LIN {X 0,Y 235.222,Z 369.249,A -85,B 0,C 180,E1 -19639.185,E2 -19639.185} C_VEL
LIN {X 0,Y 235.052,Z 370.546,A -85,B 0,C 180,E1 -19641.308,E2 -19641.308} C_VEL
LIN {X 0,Y 236.233,Z 373.828,A -85,B 0,C 180,E1 -19641.803,E2 -19641.803} C_VEL
LIN {X 0,Y 239.413,Z 381.749,A -85,B 0,C 180,E1 -19643.116,E2 -19643.116} C_VEL
LIN {X 0,Y 242.127,Z 390.64,A -85,B 0,C 180,E1 -19644.659,E2 -19644.659} C_VEL
LIN {X 0,Y 243.828,Z 398.514,A -85,B 0,C 180,E1 -19646.12,E2 -19646.12} C_VEL
LIN {X 0,Y 244.808,Z 405.816,A -85,B 0,C 180,E1 -19647.573,E2 -19647.573} C_VEL
LIN {X 0,Y 244.978,Z 410.229,A -85,B 0,C 180,E1 -19648.484,E2 -19648.484} C_VEL
LIN {X 0,Y 242.651,Z 419.105,A -85,B 0,C 180,E1 -19650.36,E2 -19650.36} C_VEL
LIN {X 0,Y 240.805,Z 425.868,A -85,B 0,C 180,E1 -19652.177,E2 -19652.177} C_VEL
LIN {X 0,Y 239.204,Z 431.176,A -85,B 0,C 180,E1 -19653.931,E2 -19653.931} C_VEL
LIN {X 0,Y 237.916,Z 435.038,A -85,B 0,C 180,E1 -19655.465,E2 -19655.465} C_VEL
LIN {X 0,Y 236.981,Z 437.92,A -85,B 0,C 180,E1 -19656.798,E2 -19656.798} C_VEL
LIN {X 0,Y 235.546,Z 441.794,A -85,B 0,C 180,E1 -19659.123,E2 -19659.123} C_VEL
LIN {X 0,Y 234.489,Z 444.579,A -85,B 0,C 180,E1 -19661.468,E2 -19661.468} C_VEL
LIN {X 0,Y 233.648,Z 446.359,A -85,B 0,C 180,E1 -19663.785,E2 -19663.785} C_VEL
LIN {X 0,Y 233.007,Z 447.26,A -85,B 0,C 180,E1 -19666.373,E2 -19666.373} C_VEL
LIN {X 0,Y 232.684,Z 447.05,A -85,B 0,C 180,E1 -19669.031,E2 -19669.031} C_VEL
LIN {X 0,Y 232.685,Z 445.653,A -85,B 0,C 180,E1 -19671.745,E2 -19671.745} C_VEL
LIN {X 0,Y 233.077,Z 442.082,A -85,B 0,C 180,E1 -19675.044,E2 -19675.044} C_VEL
LIN {X 0,Y 233.542,Z 438.663,A -85,B 0,C 180,E1 -19677.2,E2 -19677.2} C_VEL
LIN {X 0,Y 234.152,Z 434.313,A -85,B 0,C 180,E1 -19679.317,E2 -19679.317} C_VEL
LIN {X 0,Y 234.95,Z 428.913,A -85,B 0,C 180,E1 -19681.403,E2 -19681.403} C_VEL
LIN {X 0,Y 235.933,Z 422.286,A -85,B 0,C 180,E1 -19683.458,E2 -19683.458} C_VEL
LIN {X 0,Y 237.124,Z 413.918,A -85,B 0,C 180,E1 -19685.482,E2 -19685.482} C_VEL
LIN {X 0,Y 238.222,Z 405.62,A -85,B 0,C 180,E1 -19687.085,E2 -19687.085} C_VEL
LIN {X 0,Y 238.95,Z 398.643,A -85,B 0,C 180,E1 -19688.2,E2 -19688.2} C_VEL
LIN {X 0,Y 237.705,Z 390.04,A -85,B 0,C 180,E1 -19689.443,E2 -19689.443} C_VEL
LIN {X 0,Y 236.315,Z 381.565,A -85,B 0,C 180,E1 -19690.451,E2 -19690.451} C_VEL
LIN {X 0,Y 234.286,Z 371.556,A -85,B 0,C 180,E1 -19691.412,E2 -19691.412} C_VEL
LIN {X 0,Y 233.578,Z 368.098,A -85,B 0,C 180,E1 -19691.694,E2 -19691.694} C_VEL
LIN {X 0,Y 234.064,Z 364.147,A -85,B 0,C 180,E1 -19696.542,E2 -19696.542} C_VEL
LIN {X 0,Y 234.945,Z 364.031,A -85,B 0,C 180,E1 -19701.396,E2 -19701.396} C_VEL
LIN {X 0,Y 235.185,Z 364.002,A -85,B 0,C 180,E1 -19703.133,E2 -19703.133} C_VEL
LIN {X 0,Y 235.586,Z 363.954,A -85,B 0,C 180,E1 -19708.288,E2 -19708.288} C_VEL
LIN {X 0,Y 235.588,Z 363.952,A -85,B 0,C 180,E1 -19711.707,E2 -19711.707} C_VEL
LIN {X 0,Y 235.397,Z 363.973,A -85,B 0,C 180,E1 -19716.857,E2 -19716.857} C_VEL
LIN {X 0,Y 235.243,Z 363.992,A -85,B 0,C 180,E1 -19720.324,E2 -19720.324} C_VEL
LIN {X 0,Y 235.103,Z 364.013,A -85,B 0,C 180,E1 -19725.605,E2 -19725.605} C_VEL
LIN {X 0,Y 234.998,Z 364.023,A -85,B 0,C 180,E1 -19729.204,E2 -19729.204} C_VEL
LIN {X 0,Y 234.95,Z 364.029,A -85,B 0,C 180,E1 -19732.881,E2 -19732.881} C_VEL
LIN {X 0,Y 234.957,Z 364.027,A -85,B 0,C 180,E1 -19736.656,E2 -19736.656} C_VEL
LIN {X 0,Y 234.919,Z 364.032,A -85,B 0,C 180,E1 -19740.567,E2 -19740.567} C_VEL
LIN {X 0,Y 234.948,Z 364.029,A -85,B 0,C 180,E1 -19744.632,E2 -19744.632} C_VEL
LIN {X 0,Y 234.984,Z 364.026,A -85,B 0,C 180,E1 -19748.961,E2 -19748.961} C_VEL
LIN {X 0,Y 234.983,Z 364.024,A -85,B 0,C 180,E1 -19753.46,E2 -19753.46} C_VEL
LIN {X 0,Y 234.983,Z 364.025,A -85,B 0,C 180,E1 -19756.539,E2 -19756.539} C_VEL
LIN {X 0,Y 234.957,Z 364.029,A -85,B 0,C 180,E1 -19761.089,E2 -19761.089} C_VEL
LIN {X 0,Y 234.947,Z 364.03,A -85,B 0,C 180,E1 -19765.367,E2 -19765.367} C_VEL
LIN {X 0,Y 234.956,Z 364.028,A -85,B 0,C 180,E1 -19770.158,E2 -19770.158} C_VEL
LIN {X 0,Y 234.989,Z 364.025,A -85,B 0,C 180,E1 -19775.249,E2 -19775.249} C_VEL
LIN {X 0,Y 235.039,Z 364.016,A -85,B 0,C 180,E1 -19778.975,E2 -19778.975} C_VEL
LIN {X 0,Y 235.105,Z 364.01,A -85,B 0,C 180,E1 -19783.044,E2 -19783.044} C_VEL
LIN {X 0,Y 235.136,Z 364.006,A -85,B 0,C 180,E1 -19787.925,E2 -19787.925} C_VEL
LIN {X 0,Y 235.379,Z 363.976,A -85,B 0,C 180,E1 -19791.416,E2 -19791.416} C_VEL
LIN {X 0,Y 235.395,Z 363.973,A -85,B 0,C 180,E1 -19793.143,E2 -19793.143} C_VEL
LIN {X 0,Y 235.586,Z 363.952,A -85,B 0,C 180,E1 -19798.292,E2 -19798.292} C_VEL
LIN {X 0,Y 235.587,Z 363.952,A -85,B 0,C 180,E1 -19801.711,E2 -19801.711} C_VEL
LIN {X 0,Y 235.397,Z 363.973,A -85,B 0,C 180,E1 -19806.86,E2 -19806.86} C_VEL
LIN {X 0,Y 235.245,Z 363.992,A -85,B 0,C 180,E1 -19810.328,E2 -19810.328} C_VEL
LIN {X 0,Y 235.106,Z 364.013,A -85,B 0,C 180,E1 -19815.608,E2 -19815.608} C_VEL
LIN {X 0,Y 235.001,Z 364.024,A -85,B 0,C 180,E1 -19819.208,E2 -19819.208} C_VEL
LIN {X 0,Y 234.954,Z 364.028,A -85,B 0,C 180,E1 -19822.885,E2 -19822.885} C_VEL
LIN {X 0,Y 234.963,Z 364.028,A -85,B 0,C 180,E1 -19826.66,E2 -19826.66} C_VEL
LIN {X 0,Y 234.926,Z 364.031,A -85,B 0,C 180,E1 -19830.57,E2 -19830.57} C_VEL
LIN {X 0,Y 234.921,Z 364.034,A -85,B 0,C 180,E1 -19834.641,E2 -19834.641} C_VEL
LIN {X 0,Y 234.937,Z 364.032,A -85,B 0,C 180,E1 -19838.947,E2 -19838.947} C_VEL
LIN {X 0,Y 234.887,Z 364.037,A -85,B 0,C 180,E1 -19843.488,E2 -19843.488} C_VEL
LIN {X 0,Y 235.054,Z 364.178,A -85,B 0,C 180,E1 -19847.266,E2 -19847.266} C_VEL
LIN {X 0,Y 236.079,Z 369.576,A -85,B 0,C 180,E1 -19852.395,E2 -19852.395} C_VEL
LIN {X 0,Y 236.457,Z 371.989,A -85,B 0,C 180,E1 -19854.592,E2 -19854.592} C_VEL
LIN {X 0,Y 235.755,Z 373.624,A -85,B 0,C 180,E1 -19855.954,E2 -19855.954} C_VEL
LIN {X 0,Y 233.999,Z 375.327,A -85,B 0,C 180,E1 -19857.275,E2 -19857.275} C_VEL
LIN {X 0,Y 229.645,Z 378.781,A -85,B 0,C 180,E1 -19859.922,E2 -19859.922} C_VEL
LIN {X 0,Y 228.207,Z 380.506,A -85,B 0,C 180,E1 -19861.321,E2 -19861.321} C_VEL
LIN {X 0,Y 227.99,Z 381.073,A -85,B 0,C 180,E1 -19861.802,E2 -19861.802} C_VEL
LIN {X 0,Y 226.914,Z 387.476,A -85,B 0,C 180,E1 -19867.226,E2 -19867.226} C_VEL
LIN {X 0,Y 226.84,Z 388.158,A -85,B 0,C 180,E1 -19867.8,E2 -19867.8} C_VEL
LIN {X 0,Y 228.206,Z 400.804,A -85,B 0,C 180,E1 -19868.833,E2 -19868.833} C_VEL
LIN {X 0,Y 228.996,Z 409.707,A -85,B 0,C 180,E1 -19869.819,E2 -19869.819} C_VEL
LIN {X 0,Y 229.519,Z 418.83,A -85,B 0,C 180,E1 -19871.074,E2 -19871.074} C_VEL
LIN {X 0,Y 229.83,Z 426.888,A -85,B 0,C 180,E1 -19872.427,E2 -19872.427} C_VEL
LIN {X 0,Y 229.768,Z 431.689,A -85,B 0,C 180,E1 -19873.339,E2 -19873.339} C_VEL
LIN {X 0,Y 228.714,Z 438.58,A -85,B 0,C 180,E1 -19874.862,E2 -19874.862} C_VEL
LIN {X 0,Y 227.782,Z 445.123,A -85,B 0,C 180,E1 -19876.623,E2 -19876.623} C_VEL
LIN {X 0,Y 227.043,Z 450.571,A -85,B 0,C 180,E1 -19878.395,E2 -19878.395} C_VEL
LIN {X 0,Y 226.506,Z 455.12,A -85,B 0,C 180,E1 -19880.177,E2 -19880.177} C_VEL
LIN {X 0,Y 226.101,Z 458.892,A -85,B 0,C 180,E1 -19881.962,E2 -19881.962} C_VEL
LIN {X 0,Y 225.806,Z 463.172,A -85,B 0,C 180,E1 -19884.645,E2 -19884.645} C_VEL
LIN {X 0,Y 225.811,Z 465.347,A -85,B 0,C 180,E1 -19886.434,E2 -19886.434} C_VEL
LIN {X 0,Y 225.863,Z 466.928,A -85,B 0,C 180,E1 -19888.219,E2 -19888.219} C_VEL
LIN {X 0,Y 225.879,Z 467.899,A -85,B 0,C 180,E1 -19890.002,E2 -19890.002} C_VEL
LIN {X 0,Y 225.837,Z 468.378,A -85,B 0,C 180,E1 -19891.786,E2 -19891.786} C_VEL
LIN {X 0,Y 225.724,Z 468.081,A -85,B 0,C 180,E1 -19894.898,E2 -19894.898} C_VEL
LIN {X 0,Y 225.925,Z 466.884,A -85,B 0,C 180,E1 -19897.15,E2 -19897.15} C_VEL
LIN {X 0,Y 226.536,Z 464.45,A -85,B 0,C 180,E1 -19899.827,E2 -19899.827} C_VEL
LIN {X 0,Y 227.599,Z 460.723,A -85,B 0,C 180,E1 -19902.485,E2 -19902.485} C_VEL
LIN {X 0,Y 228.613,Z 457.567,A -85,B 0,C 180,E1 -19904.239,E2 -19904.239} C_VEL
LIN {X 0,Y 230.195,Z 452.594,A -85,B 0,C 180,E1 -19906.406,E2 -19906.406} C_VEL
LIN {X 0,Y 232.154,Z 446.383,A -85,B 0,C 180,E1 -19908.536,E2 -19908.536} C_VEL
LIN {X 0,Y 233.868,Z 440.38,A -85,B 0,C 180,E1 -19910.22,E2 -19910.22} C_VEL
LIN {X 0,Y 234.91,Z 434.608,A -85,B 0,C 180,E1 -19911.639,E2 -19911.639} C_VEL
LIN {X 0,Y 235.513,Z 426.948,A -85,B 0,C 180,E1 -19913.293,E2 -19913.293} C_VEL
LIN {X 0,Y 235.484,Z 419.713,A -85,B 0,C 180,E1 -19914.7,E2 -19914.7} C_VEL
LIN {X 0,Y 234.896,Z 411.306,A -85,B 0,C 180,E1 -19916.155,E2 -19916.155} C_VEL
LIN {X 0,Y 233.253,Z 401.765,A -85,B 0,C 180,E1 -19917.679,E2 -19917.679} C_VEL
LIN {X 0,Y 230.783,Z 391.922,A -85,B 0,C 180,E1 -19919.135,E2 -19919.135} C_VEL
LIN {X 0,Y 229.176,Z 386.225,A -85,B 0,C 180,E1 -19919.919,E2 -19919.919} C_VEL
LIN {X 0,Y 229.114,Z 385.693,A -85,B 0,C 180,E1 -19919.974,E2 -19919.974} C_VEL
LIN {X 0,Y 230.038,Z 382.099,A -85,B 0,C 180,E1 -19923.364,E2 -19923.364} C_VEL
LIN {X 0,Y 230.33,Z 380.041,A -85,B 0,C 180,E1 -19925.435,E2 -19925.435} C_VEL
LIN {X 0,Y 230.126,Z 378.022,A -85,B 0,C 180,E1 -19927.649,E2 -19927.649} C_VEL
LIN {X 0,Y 229.807,Z 375.884,A -85,B 0,C 180,E1 -19930.131,E2 -19930.131} C_VEL
LIN {X 0,Y 229.106,Z 372.001,A -85,B 0,C 180,E1 -19935.125,E2 -19935.125} C_VEL
LIN {X 0,Y 228.556,Z 368.903,A -85,B 0,C 180,E1 -19939.777,E2 -19939.777} C_VEL
LIN {X 0,Y 228.267,Z 366.929,A -85,B 0,C 180,E1 -19943.181,E2 -19943.181} C_VEL
LIN {X 0,Y 227.952,Z 365.343,A -85,B 0,C 180,E1 -19946.353,E2 -19946.353} C_VEL
LIN {X 0,Y 227.906,Z 364.908,A -85,B 0,C 180,E1 -19949.709,E2 -19949.709} C_VEL
LIN {X 0,Y 227.938,Z 364.906,A -85,B 0,C 180,E1 -19954.425,E2 -19954.425} C_VEL
LIN {X 0,Y 227.972,Z 364.9,A -85,B 0,C 180,E1 -19958.286,E2 -19958.286} C_VEL
LIN {X 0,Y 228.044,Z 364.891,A -85,B 0,C 180,E1 -19962.825,E2 -19962.825} C_VEL
LIN {X 0,Y 228.077,Z 364.887,A -85,B 0,C 180,E1 -19967.542,E2 -19967.542} C_VEL
LIN {X 0,Y 228.268,Z 364.864,A -85,B 0,C 180,E1 -19971.143,E2 -19971.143} C_VEL
LIN {X 0,Y 228.318,Z 364.859,A -85,B 0,C 180,E1 -19972.926,E2 -19972.926} C_VEL
LIN {X 0,Y 228.558,Z 364.824,A -85,B 0,C 180,E1 -19978.236,E2 -19978.236} C_VEL
LIN {X 0,Y 228.56,Z 364.825,A -85,B 0,C 180,E1 -19981.76,E2 -19981.76} C_VEL
LIN {X 0,Y 228.324,Z 364.857,A -85,B 0,C 180,E1 -19987.071,E2 -19987.071} C_VEL
LIN {X 0,Y 228.346,Z 366.209,A -85,B 0,C 180,E1 -19990.64,E2 -19990.64} C_VEL
LIN {X 0,Y 228.451,Z 367.882,A -85,B 0,C 180,E1 -19994.245,E2 -19994.245} C_VEL
LIN {X 0,Y 228.33,Z 369.822,A -85,B 0,C 180,E1 -19997.925,E2 -19997.925} C_VEL
LIN {X 0,Y 228.168,Z 371.16,A -85,B 0,C 180,E1 -19999.979,E2 -19999.979} C_VEL
LIN {X 0,Y 229.395,Z 374.35,A -85,B 0,C 180,E1 -20000.51,E2 -20000.51} C_VEL
LIN {X 0,Y 232.806,Z 382.459,A -85,B 0,C 180,E1 -20002.004,E2 -20002.004} C_VEL
LIN {X 0,Y 235.293,Z 390.144,A -85,B 0,C 180,E1 -20003.428,E2 -20003.428} C_VEL
LIN {X 0,Y 237.051,Z 397.629,A -85,B 0,C 180,E1 -20004.872,E2 -20004.872} C_VEL
LIN {X 0,Y 238.198,Z 405.563,A -85,B 0,C 180,E1 -20006.526,E2 -20006.526} C_VEL
LIN {X 0,Y 238.498,Z 411.568,A -85,B 0,C 180,E1 -20007.864,E2 -20007.864} C_VEL
LIN {X 0,Y 236.344,Z 419.358,A -85,B 0,C 180,E1 -20009.563,E2 -20009.563} C_VEL
LIN {X 0,Y 234.455,Z 425.798,A -85,B 0,C 180,E1 -20011.313,E2 -20011.313} C_VEL
LIN {X 0,Y 232.512,Z 431.916,A -85,B 0,C 180,E1 -20013.386,E2 -20013.386} C_VEL
LIN {X 0,Y 230.882,Z 436.503,A -85,B 0,C 180,E1 -20015.332,E2 -20015.332} C_VEL
LIN {X 0,Y 229.205,Z 441.046,A -85,B 0,C 180,E1 -20017.822,E2 -20017.822} C_VEL
LIN {X 0,Y 227.864,Z 444.363,A -85,B 0,C 180,E1 -20020.366,E2 -20020.366} C_VEL
LIN {X 0,Y 226.802,Z 446.504,A -85,B 0,C 180,E1 -20022.975,E2 -20022.975} C_VEL
LIN {X 0,Y 226.075,Z 447.547,A -85,B 0,C 180,E1 -20025.64,E2 -20025.64} C_VEL
LIN {X 0,Y 225.655,Z 447.49,A -85,B 0,C 180,E1 -20028.369,E2 -20028.369} C_VEL
LIN {X 0,Y 225.587,Z 446.09,A -85,B 0,C 180,E1 -20031.456,E2 -20031.456} C_VEL
LIN {X 0,Y 225.798,Z 443.719,A -85,B 0,C 180,E1 -20034.019,E2 -20034.019} C_VEL
LIN {X 0,Y 226.184,Z 441.098,A -85,B 0,C 180,E1 -20035.99,E2 -20035.99} C_VEL
LIN {X 0,Y 226.86,Z 436.252,A -85,B 0,C 180,E1 -20038.678,E2 -20038.678} C_VEL
LIN {X 0,Y 227.618,Z 431.025,A -85,B 0,C 180,E1 -20040.9,E2 -20040.9} C_VEL
LIN {X 0,Y 228.344,Z 426.452,A -85,B 0,C 180,E1 -20042.503,E2 -20042.503} C_VEL
LIN {X 0,Y 229.41,Z 419.09,A -85,B 0,C 180,E1 -20044.601,E2 -20044.601} C_VEL
LIN {X 0,Y 230.518,Z 411.603,A -85,B 0,C 180,E1 -20046.324,E2 -20046.324} C_VEL
LIN {X 0,Y 231.701,Z 402.878,A -85,B 0,C 180,E1 -20047.951,E2 -20047.951} C_VEL
LIN {X 0,Y 232.001,Z 399.711,A -85,B 0,C 180,E1 -20048.448,E2 -20048.448} C_VEL
LIN {X 0,Y 230.807,Z 391.249,A -85,B 0,C 180,E1 -20049.733,E2 -20049.733} C_VEL
LIN {X 0,Y 229.483,Z 382.947,A -85,B 0,C 180,E1 -20050.776,E2 -20050.776} C_VEL
LIN {X 0,Y 227.536,Z 373.182,A -85,B 0,C 180,E1 -20051.774,E2 -20051.774} C_VEL
LIN {X 0,Y 226.56,Z 368.36,A -85,B 0,C 180,E1 -20052.218,E2 -20052.218} C_VEL
LIN {X 0,Y 227.018,Z 365.024,A -85,B 0,C 180,E1 -20056.572,E2 -20056.572} C_VEL
LIN {X 0,Y 227.87,Z 364.912,A -85,B 0,C 180,E1 -20061.127,E2 -20061.127} C_VEL
LIN {X 0,Y 228.099,Z 364.885,A -85,B 0,C 180,E1 -20062.918,E2 -20062.918} C_VEL
LIN {X 0,Y 228.544,Z 364.832,A -85,B 0,C 180,E1 -20068.236,E2 -20068.236} C_VEL
LIN {X 0,Y 228.547,Z 364.83,A -85,B 0,C 180,E1 -20071.76,E2 -20071.76} C_VEL
LIN {X 0,Y 228.349,Z 364.851,A -85,B 0,C 180,E1 -20077.069,E2 -20077.069} C_VEL
LIN {X 0,Y 228.162,Z 364.873,A -85,B 0,C 180,E1 -20080.648,E2 -20080.648} C_VEL
LIN {X 0,Y 228.047,Z 364.891,A -85,B 0,C 180,E1 -20086.1,E2 -20086.1} C_VEL
LIN {X 0,Y 227.932,Z 364.904,A -85,B 0,C 180,E1 -20089.824,E2 -20089.824} C_VEL
LIN {X 0,Y 227.903,Z 364.911,A -85,B 0,C 180,E1 -20093.631,E2 -20093.631} C_VEL
LIN {X 0,Y 227.873,Z 364.911,A -85,B 0,C 180,E1 -20097.554,E2 -20097.554} C_VEL
LIN {X 0,Y 227.86,Z 364.915,A -85,B 0,C 180,E1 -20101.621,E2 -20101.621} C_VEL
LIN {X 0,Y 227.89,Z 364.906,A -85,B 0,C 180,E1 -20105.867,E2 -20105.867} C_VEL
LIN {X 0,Y 227.905,Z 364.907,A -85,B 0,C 180,E1 -20110.356,E2 -20110.356} C_VEL
LIN {X 0,Y 227.907,Z 364.907,A -85,B 0,C 180,E1 -20114.829,E2 -20114.829} C_VEL
LIN {X 0,Y 227.922,Z 364.905,A -85,B 0,C 180,E1 -20117.731,E2 -20117.731} C_VEL
LIN {X 0,Y 227.868,Z 364.91,A -85,B 0,C 180,E1 -20121.916,E2 -20121.916} C_VEL
LIN {X 0,Y 227.877,Z 364.911,A -85,B 0,C 180,E1 -20126.373,E2 -20126.373} C_VEL
LIN {X 0,Y 227.906,Z 364.908,A -85,B 0,C 180,E1 -20130.438,E2 -20130.438} C_VEL
LIN {X 0,Y 227.922,Z 364.907,A -85,B 0,C 180,E1 -20134.427,E2 -20134.427} C_VEL
LIN {X 0,Y 227.999,Z 364.897,A -85,B 0,C 180,E1 -20138.293,E2 -20138.293} C_VEL
LIN {X 0,Y 228.034,Z 364.892,A -85,B 0,C 180,E1 -20142.818,E2 -20142.818} C_VEL
LIN {X 0,Y 228.083,Z 364.882,A -85,B 0,C 180,E1 -20147.546,E2 -20147.546} C_VEL
LIN {X 0,Y 228.314,Z 364.856,A -85,B 0,C 180,E1 -20151.148,E2 -20151.148} C_VEL
LIN {X 0,Y 228.347,Z 364.852,A -85,B 0,C 180,E1 -20152.93,E2 -20152.93} C_VEL
LIN {X 0,Y 228.545,Z 364.829,A -85,B 0,C 180,E1 -20158.24,E2 -20158.24} C_VEL
LIN {X 0,Y 228.546,Z 364.83,A -85,B 0,C 180,E1 -20161.764,E2 -20161.764} C_VEL
LIN {X 0,Y 228.349,Z 364.851,A -85,B 0,C 180,E1 -20167.073,E2 -20167.073} C_VEL
LIN {X 0,Y 228.159,Z 364.874,A -85,B 0,C 180,E1 -20170.652,E2 -20170.652} C_VEL
LIN {X 0,Y 228.057,Z 364.887,A -85,B 0,C 180,E1 -20174.274,E2 -20174.274} C_VEL
LIN {X 0,Y 227.996,Z 364.896,A -85,B 0,C 180,E1 -20177.956,E2 -20177.956} C_VEL
LIN {X 0,Y 227.923,Z 364.903,A -85,B 0,C 180,E1 -20182.332,E2 -20182.332} C_VEL
LIN {X 0,Y 227.937,Z 364.903,A -85,B 0,C 180,E1 -20186.605,E2 -20186.605} C_VEL
LIN {X 0,Y 227.903,Z 364.905,A -85,B 0,C 180,E1 -20190.299,E2 -20190.299} C_VEL
LIN {X 0,Y 227.871,Z 364.912,A -85,B 0,C 180,E1 -20193.723,E2 -20193.723} C_VEL
LIN {X 0,Y 227.839,Z 364.913,A -85,B 0,C 180,E1 -20198.094,E2 -20198.094} C_VEL
LIN {X 0,Y 227.809,Z 364.921,A -85,B 0,C 180,E1 -20202.745,E2 -20202.745} C_VEL
LIN {X 0,Y 228.01,Z 365.07,A -85,B 0,C 180,E1 -20207.116,E2 -20207.116} C_VEL
LIN {X 0,Y 228.965,Z 370.174,A -85,B 0,C 180,E1 -20212.132,E2 -20212.132} C_VEL
LIN {X 0,Y 229.383,Z 372.742,A -85,B 0,C 180,E1 -20214.543,E2 -20214.543} C_VEL
LIN {X 0,Y 229.319,Z 374.955,A -85,B 0,C 180,E1 -20216.523,E2 -20216.523} C_VEL
LIN {X 0,Y 228.666,Z 378.252,A -85,B 0,C 180,E1 -20219.383,E2 -20219.383} C_VEL
LIN {X 0,Y 227.99,Z 381.073,A -85,B 0,C 180,E1 -20221.802,E2 -20221.802} C_VEL
LIN {X 0,Y 227.071,Z 382.206,A -85,B 0,C 180,E1 -20222.731,E2 -20222.731} C_VEL
LIN {X 0,Y 223.903,Z 384.061,A -85,B 0,C 180,E1 -20224.164,E2 -20224.164} C_VEL
LIN {X 0,Y 220.762,Z 385.925,A -85,B 0,C 180,E1 -20225.635,E2 -20225.635} C_VEL
LIN {X 0,Y 219.924,Z 387.076,A -85,B 0,C 180,E1 -20226.607,E2 -20226.607} C_VEL
LIN {X 0,Y 219.813,Z 387.82,A -85,B 0,C 180,E1 -20227.255,E2 -20227.255} C_VEL
LIN {X 0,Y 221.23,Z 400.594,A -85,B 0,C 180,E1 -20228.37,E2 -20228.37} C_VEL
LIN {X 0,Y 221.994,Z 409.762,A -85,B 0,C 180,E1 -20229.428,E2 -20229.428} C_VEL
LIN {X 0,Y 222.418,Z 418.033,A -85,B 0,C 180,E1 -20230.597,E2 -20230.597} C_VEL
LIN {X 0,Y 222.746,Z 425.393,A -85,B 0,C 180,E1 -20231.849,E2 -20231.849} C_VEL
LIN {X 0,Y 222.753,Z 431.444,A -85,B 0,C 180,E1 -20233.034,E2 -20233.034} C_VEL
LIN {X 0,Y 221.554,Z 439.172,A -85,B 0,C 180,E1 -20234.831,E2 -20234.831} C_VEL
LIN {X 0,Y 220.638,Z 445.564,A -85,B 0,C 180,E1 -20236.65,E2 -20236.65} C_VEL
LIN {X 0,Y 219.879,Z 450.875,A -85,B 0,C 180,E1 -20238.479,E2 -20238.479} C_VEL
LIN {X 0,Y 219.275,Z 456.267,A -85,B 0,C 180,E1 -20240.781,E2 -20240.781} C_VEL
LIN {X 0,Y 218.935,Z 459.744,A -85,B 0,C 180,E1 -20242.625,E2 -20242.625} C_VEL
LIN {X 0,Y 218.709,Z 463.215,A -85,B 0,C 180,E1 -20244.987,E2 -20244.987} C_VEL
LIN {X 0,Y 218.714,Z 464.816,A -85,B 0,C 180,E1 -20246.318,E2 -20246.318} C_VEL
LIN {X 0,Y 218.795,Z 466.416,A -85,B 0,C 180,E1 -20248.162,E2 -20248.162} C_VEL
LIN {X 0,Y 218.81,Z 467.454,A -85,B 0,C 180,E1 -20250.002,E2 -20250.002} C_VEL
LIN {X 0,Y 218.743,Z 468.003,A -85,B 0,C 180,E1 -20251.844,E2 -20251.844} C_VEL
LIN {X 0,Y 218.623,Z 467.847,A -85,B 0,C 180,E1 -20254.748,E2 -20254.748} C_VEL
LIN {X 0,Y 218.862,Z 466.661,A -85,B 0,C 180,E1 -20257.382,E2 -20257.382} C_VEL
LIN {X 0,Y 219.248,Z 465.19,A -85,B 0,C 180,E1 -20259.225,E2 -20259.225} C_VEL
LIN {X 0,Y 220.222,Z 462.044,A -85,B 0,C 180,E1 -20261.974,E2 -20261.974} C_VEL
LIN {X 0,Y 221.724,Z 457.649,A -85,B 0,C 180,E1 -20264.692,E2 -20264.692} C_VEL
LIN {X 0,Y 223.729,Z 451.653,A -85,B 0,C 180,E1 -20267.365,E2 -20267.365} C_VEL
LIN {X 0,Y 225.915,Z 445.318,A -85,B 0,C 180,E1 -20269.54,E2 -20269.54} C_VEL
LIN {X 0,Y 227.601,Z 439.223,A -85,B 0,C 180,E1 -20271.276,E2 -20271.276} C_VEL
LIN {X 0,Y 228.523,Z 433.646,A -85,B 0,C 180,E1 -20272.685,E2 -20272.685} C_VEL
LIN {X 0,Y 229.124,Z 425.632,A -85,B 0,C 180,E1 -20274.464,E2 -20274.464} C_VEL
LIN {X 0,Y 228.971,Z 417.582,A -85,B 0,C 180,E1 -20276.059,E2 -20276.059} C_VEL
LIN {X 0,Y 228.147,Z 409.462,A -85,B 0,C 180,E1 -20277.523,E2 -20277.523} C_VEL
LIN {X 0,Y 226.749,Z 401.44,A -85,B 0,C 180,E1 -20278.882,E2 -20278.882} C_VEL
LIN {X 0,Y 224.445,Z 392.356,A -85,B 0,C 180,E1 -20280.335,E2 -20280.335} C_VEL
LIN {X 0,Y 223.067,Z 387.959,A -85,B 0,C 180,E1 -20281.04,E2 -20281.04} C_VEL
LIN {X 0,Y 222.454,Z 385.249,A -85,B 0,C 180,E1 -20281.397,E2 -20281.397} C_VEL
LIN {X 0,Y 223.247,Z 382.117,A -85,B 0,C 180,E1 -20284.52,E2 -20284.52} C_VEL
LIN {X 0,Y 223.078,Z 378.973,A -85,B 0,C 180,E1 -20288.035,E2 -20288.035} C_VEL
LIN {X 0,Y 222.606,Z 376.133,A -85,B 0,C 180,E1 -20291.532,E2 -20291.532} C_VEL
LIN {X 0,Y 222.029,Z 372.99,A -85,B 0,C 180,E1 -20295.861,E2 -20295.861} C_VEL
LIN {X 0,Y 221.571,Z 369.972,A -85,B 0,C 180,E1 -20300.624,E2 -20300.624} C_VEL
LIN {X 0,Y 221.397,Z 368.697,A -85,B 0,C 180,E1 -20302.904,E2 -20302.904} C_VEL
LIN {X 0,Y 220.961,Z 366.628,A -85,B 0,C 180,E1 -20307.266,E2 -20307.266} C_VEL
LIN {X 0,Y 220.844,Z 365.789,A -85,B 0,C 180,E1 -20309.389,E2 -20309.389} C_VEL
LIN {X 0,Y 220.904,Z 365.781,A -85,B 0,C 180,E1 -20313.549,E2 -20313.549} C_VEL
LIN {X 0,Y 220.888,Z 365.784,A -85,B 0,C 180,E1 -20317.553,E2 -20317.553} C_VEL
LIN {X 0,Y 220.994,Z 365.769,A -85,B 0,C 180,E1 -20322.57,E2 -20322.57} C_VEL
LIN {X 0,Y 221.017,Z 365.767,A -85,B 0,C 180,E1 -20327.137,E2 -20327.137} C_VEL
LIN {X 0,Y 221.207,Z 365.743,A -85,B 0,C 180,E1 -20330.858,E2 -20330.858} C_VEL
LIN {X 0,Y 221.133,Z 365.754,A -85,B 0,C 180,E1 -20334.527,E2 -20334.527} C_VEL
LIN {X 0,Y 221.516,Z 365.701,A -85,B 0,C 180,E1 -20338.18,E2 -20338.18} C_VEL
LIN {X 0,Y 221.518,Z 365.703,A -85,B 0,C 180,E1 -20341.816,E2 -20341.816} C_VEL
LIN {X 0,Y 221.141,Z 365.75,A -85,B 0,C 180,E1 -20345.469,E2 -20345.469} C_VEL
LIN {X 0,Y 221.349,Z 366.292,A -85,B 0,C 180,E1 -20347.295,E2 -20347.295} C_VEL
LIN {X 0,Y 221.402,Z 367.783,A -85,B 0,C 180,E1 -20350.978,E2 -20350.978} C_VEL
LIN {X 0,Y 221.476,Z 369.468,A -85,B 0,C 180,E1 -20354.704,E2 -20354.704} C_VEL
LIN {X 0,Y 221.277,Z 371.427,A -85,B 0,C 180,E1 -20358.468,E2 -20358.468} C_VEL
LIN {X 0,Y 222.475,Z 374.707,A -85,B 0,C 180,E1 -20359.071,E2 -20359.071} C_VEL
LIN {X 0,Y 225.705,Z 381.835,A -85,B 0,C 180,E1 -20360.504,E2 -20360.504} C_VEL
LIN {X 0,Y 228.504,Z 389.954,A -85,B 0,C 180,E1 -20362.131,E2 -20362.131} C_VEL
LIN {X 0,Y 230.555,Z 398.263,A -85,B 0,C 180,E1 -20363.862,E2 -20363.862} C_VEL
LIN {X 0,Y 231.717,Z 406.222,A -85,B 0,C 180,E1 -20365.605,E2 -20365.605} C_VEL
LIN {X 0,Y 232.032,Z 413.115,A -85,B 0,C 180,E1 -20367.24,E2 -20367.24} C_VEL
LIN {X 0,Y 230.006,Z 419.935,A -85,B 0,C 180,E1 -20368.782,E2 -20368.782} C_VEL
LIN {X 0,Y 228.178,Z 425.792,A -85,B 0,C 180,E1 -20370.408,E2 -20370.408} C_VEL
LIN {X 0,Y 226.305,Z 431.357,A -85,B 0,C 180,E1 -20372.302,E2 -20372.302} C_VEL
LIN {X 0,Y 224.548,Z 436.08,A -85,B 0,C 180,E1 -20374.287,E2 -20374.287} C_VEL
LIN {X 0,Y 223.19,Z 439.612,A -85,B 0,C 180,E1 -20376.123,E2 -20376.123} C_VEL
LIN {X 0,Y 221.585,Z 443.313,A -85,B 0,C 180,E1 -20378.653,E2 -20378.653} C_VEL
LIN {X 0,Y 220.822,Z 445.045,A -85,B 0,C 180,E1 -20380.193,E2 -20380.193} C_VEL
LIN {X 0,Y 219.807,Z 446.922,A -85,B 0,C 180,E1 -20382.657,E2 -20382.657} C_VEL
LIN {X 0,Y 219.1,Z 447.876,A -85,B 0,C 180,E1 -20385.112,E2 -20385.112} C_VEL
LIN {X 0,Y 218.632,Z 447.926,A -85,B 0,C 180,E1 -20387.672,E2 -20387.672} C_VEL
LIN {X 0,Y 218.449,Z 446.85,A -85,B 0,C 180,E1 -20390.542,E2 -20390.542} C_VEL
LIN {X 0,Y 218.626,Z 444.524,A -85,B 0,C 180,E1 -20393.477,E2 -20393.477} C_VEL
LIN {X 0,Y 219.166,Z 440.644,A -85,B 0,C 180,E1 -20396.481,E2 -20396.481} C_VEL
LIN {X 0,Y 219.743,Z 436.737,A -85,B 0,C 180,E1 -20398.684,E2 -20398.684} C_VEL
LIN {X 0,Y 220.529,Z 431.478,A -85,B 0,C 180,E1 -20401,E2 -20401} C_VEL
LIN {X 0,Y 221.338,Z 426.62,A -85,B 0,C 180,E1 -20402.751,E2 -20402.751} C_VEL
LIN {X 0,Y 222.304,Z 419.915,A -85,B 0,C 180,E1 -20404.733,E2 -20404.733} C_VEL
LIN {X 0,Y 223.422,Z 412.866,A -85,B 0,C 180,E1 -20406.433,E2 -20406.433} C_VEL
LIN {X 0,Y 224.45,Z 405.347,A -85,B 0,C 180,E1 -20407.927,E2 -20407.927} C_VEL
LIN {X 0,Y 225.017,Z 400.819,A -85,B 0,C 180,E1 -20408.708,E2 -20408.708} C_VEL
LIN {X 0,Y 223.911,Z 392.463,A -85,B 0,C 180,E1 -20410.039,E2 -20410.039} C_VEL
LIN {X 0,Y 222.654,Z 384.338,A -85,B 0,C 180,E1 -20411.121,E2 -20411.121} C_VEL
LIN {X 0,Y 220.778,Z 374.728,A -85,B 0,C 180,E1 -20412.156,E2 -20412.156} C_VEL
LIN {X 0,Y 219.529,Z 368.694,A -85,B 0,C 180,E1 -20412.712,E2 -20412.712} C_VEL
LIN {X 0,Y 219.934,Z 365.908,A -85,B 0,C 180,E1 -20416.367,E2 -20416.367} C_VEL
LIN {X 0,Y 220.763,Z 365.799,A -85,B 0,C 180,E1 -20420.839,E2 -20420.839} C_VEL
LIN {X 0,Y 221.018,Z 365.768,A -85,B 0,C 180,E1 -20422.69,E2 -20422.69} C_VEL
LIN {X 0,Y 221.501,Z 365.71,A -85,B 0,C 180,E1 -20428.179,E2 -20428.179} C_VEL
LIN {X 0,Y 221.505,Z 365.707,A -85,B 0,C 180,E1 -20431.816,E2 -20431.816} C_VEL
LIN {X 0,Y 221.302,Z 365.73,A -85,B 0,C 180,E1 -20437.296,E2 -20437.296} C_VEL
LIN {X 0,Y 221.107,Z 365.751,A -85,B 0,C 180,E1 -20440.992,E2 -20440.992} C_VEL
LIN {X 0,Y 221.006,Z 365.766,A -85,B 0,C 180,E1 -20446.628,E2 -20446.628} C_VEL
LIN {X 0,Y 220.882,Z 365.779,A -85,B 0,C 180,E1 -20450.484,E2 -20450.484} C_VEL
LIN {X 0,Y 220.856,Z 365.785,A -85,B 0,C 180,E1 -20454.433,E2 -20454.433} C_VEL
LIN {X 0,Y 220.824,Z 365.786,A -85,B 0,C 180,E1 -20458.512,E2 -20458.512} C_VEL
LIN {X 0,Y 220.812,Z 365.791,A -85,B 0,C 180,E1 -20462.754,E2 -20462.754} C_VEL
LIN {X 0,Y 220.855,Z 365.786,A -85,B 0,C 180,E1 -20467.297,E2 -20467.297} C_VEL
LIN {X 0,Y 220.866,Z 365.783,A -85,B 0,C 180,E1 -20471.927,E2 -20471.927} C_VEL
LIN {X 0,Y 220.862,Z 365.783,A -85,B 0,C 180,E1 -20475.572,E2 -20475.572} C_VEL
LIN {X 0,Y 220.848,Z 365.786,A -85,B 0,C 180,E1 -20479.791,E2 -20479.791} C_VEL
LIN {X 0,Y 220.826,Z 365.789,A -85,B 0,C 180,E1 -20482.796,E2 -20482.796} C_VEL
LIN {X 0,Y 220.811,Z 365.791,A -85,B 0,C 180,E1 -20487.246,E2 -20487.246} C_VEL
LIN {X 0,Y 220.824,Z 365.786,A -85,B 0,C 180,E1 -20491.487,E2 -20491.487} C_VEL
LIN {X 0,Y 220.871,Z 365.783,A -85,B 0,C 180,E1 -20495.568,E2 -20495.568} C_VEL
LIN {X 0,Y 220.914,Z 365.774,A -85,B 0,C 180,E1 -20499.518,E2 -20499.518} C_VEL
LIN {X 0,Y 221.014,Z 365.765,A -85,B 0,C 180,E1 -20503.372,E2 -20503.372} C_VEL
LIN {X 0,Y 221.106,Z 365.752,A -85,B 0,C 180,E1 -20509.008,E2 -20509.008} C_VEL
LIN {X 0,Y 221.3,Z 365.73,A -85,B 0,C 180,E1 -20512.704,E2 -20512.704} C_VEL
LIN {X 0,Y 221.503,Z 365.707,A -85,B 0,C 180,E1 -20518.184,E2 -20518.184} C_VEL
LIN {X 0,Y 221.504,Z 365.707,A -85,B 0,C 180,E1 -20521.82,E2 -20521.82} C_VEL
LIN {X 0,Y 221.302,Z 365.73,A -85,B 0,C 180,E1 -20527.3,E2 -20527.3} C_VEL
LIN {X 0,Y 221.103,Z 365.753,A -85,B 0,C 180,E1 -20530.996,E2 -20530.996} C_VEL
LIN {X 0,Y 221.009,Z 365.766,A -85,B 0,C 180,E1 -20536.632,E2 -20536.632} C_VEL
LIN {X 0,Y 220.885,Z 365.778,A -85,B 0,C 180,E1 -20540.488,E2 -20540.488} C_VEL
LIN {X 0,Y 220.861,Z 365.784,A -85,B 0,C 180,E1 -20544.437,E2 -20544.437} C_VEL
LIN {X 0,Y 220.831,Z 365.786,A -85,B 0,C 180,E1 -20548.516,E2 -20548.516} C_VEL
LIN {X 0,Y 220.812,Z 365.792,A -85,B 0,C 180,E1 -20552.759,E2 -20552.759} C_VEL
LIN {X 0,Y 220.805,Z 365.791,A -85,B 0,C 180,E1 -20557.281,E2 -20557.281} C_VEL
LIN {X 0,Y 220.767,Z 365.796,A -85,B 0,C 180,E1 -20561.955,E2 -20561.955} C_VEL
LIN {X 0,Y 220.945,Z 365.985,A -85,B 0,C 180,E1 -20567.023,E2 -20567.023} C_VEL
LIN {X 0,Y 221.588,Z 369.531,A -85,B 0,C 180,E1 -20570.633,E2 -20570.633} C_VEL
LIN {X 0,Y 222.309,Z 373.175,A -85,B 0,C 180,E1 -20574.212,E2 -20574.212} C_VEL
LIN {X 0,Y 222.267,Z 375.535,A -85,B 0,C 180,E1 -20576.407,E2 -20576.407} C_VEL
LIN {X 0,Y 221.23,Z 380.117,A -85,B 0,C 180,E1 -20580.504,E2 -20580.504} C_VEL
LIN {X 0,Y 220.088,Z 385.78,A -85,B 0,C 180,E1 -20585.476,E2 -20585.476} C_VEL
LIN {X 0,Y 219.924,Z 387.076,A -85,B 0,C 180,E1 -20586.607,E2 -20586.607} C_VEL
LIN {X 0,Y 219.839,Z 388.555,A -85,B 0,C 180,E1 -20587.121,E2 -20587.121} C_VEL
LIN {X 0,Y 219.734,Z 391.899,A -85,B 0,C 180,E1 -20587.534,E2 -20587.534} C_VEL
LIN {X 0,Y 218.798,Z 401.426,A -85,B 0,C 180,E1 -20588.28,E2 -20588.28} C_VEL
LIN {X 0,Y 215.763,Z 412.226,A -85,B 0,C 180,E1 -20589.32,E2 -20589.32} C_VEL
LIN {X 0,Y 215.338,Z 415.796,A -85,B 0,C 180,E1 -20589.865,E2 -20589.865} C_VEL
LIN {X 0,Y 215.705,Z 425.143,A -85,B 0,C 180,E1 -20591.481,E2 -20591.481} C_VEL
LIN {X 0,Y 215.624,Z 432.219,A -85,B 0,C 180,E1 -20592.944,E2 -20592.944} C_VEL
LIN {X 0,Y 214.397,Z 439.76,A -85,B 0,C 180,E1 -20594.8,E2 -20594.8} C_VEL
LIN {X 0,Y 213.504,Z 445.999,A -85,B 0,C 180,E1 -20596.681,E2 -20596.681} C_VEL
LIN {X 0,Y 212.742,Z 451.171,A -85,B 0,C 180,E1 -20598.57,E2 -20598.57} C_VEL
LIN {X 0,Y 212.247,Z 455.484,A -85,B 0,C 180,E1 -20600.473,E2 -20600.473} C_VEL
LIN {X 0,Y 211.786,Z 460.566,A -85,B 0,C 180,E1 -20603.333,E2 -20603.333} C_VEL
LIN {X 0,Y 211.621,Z 464.24,A -85,B 0,C 180,E1 -20606.194,E2 -20606.194} C_VEL
LIN {X 0,Y 211.726,Z 465.884,A -85,B 0,C 180,E1 -20608.1,E2 -20608.1} C_VEL
LIN {X 0,Y 211.743,Z 466.999,A -85,B 0,C 180,E1 -20610.002,E2 -20610.002} C_VEL
LIN {X 0,Y 211.65,Z 467.624,A -85,B 0,C 180,E1 -20611.905,E2 -20611.905} C_VEL
LIN {X 0,Y 211.54,Z 467.604,A -85,B 0,C 180,E1 -20614.648,E2 -20614.648} C_VEL
LIN {X 0,Y 211.823,Z 466.441,A -85,B 0,C 180,E1 -20617.629,E2 -20617.629} C_VEL
LIN {X 0,Y 212.234,Z 465.051,A -85,B 0,C 180,E1 -20619.533,E2 -20619.533} C_VEL
LIN {X 0,Y 213.276,Z 461.989,A -85,B 0,C 180,E1 -20622.37,E2 -20622.37} C_VEL
LIN {X 0,Y 214.847,Z 457.704,A -85,B 0,C 180,E1 -20625.173,E2 -20625.173} C_VEL
LIN {X 0,Y 216.974,Z 451.937,A -85,B 0,C 180,E1 -20627.924,E2 -20627.924} C_VEL
LIN {X 0,Y 219.266,Z 445.758,A -85,B 0,C 180,E1 -20630.157,E2 -20630.157} C_VEL
LIN {X 0,Y 221.022,Z 439.816,A -85,B 0,C 180,E1 -20631.942,E2 -20631.942} C_VEL
LIN {X 0,Y 222.18,Z 432.74,A -85,B 0,C 180,E1 -20633.795,E2 -20633.795} C_VEL
LIN {X 0,Y 222.671,Z 425.486,A -85,B 0,C 180,E1 -20635.472,E2 -20635.472} C_VEL
LIN {X 0,Y 222.576,Z 417.744,A -85,B 0,C 180,E1 -20637.09,E2 -20637.09} C_VEL
LIN {X 0,Y 221.813,Z 409.714,A -85,B 0,C 180,E1 -20638.638,E2 -20638.638} C_VEL
LIN {X 0,Y 220.396,Z 401.474,A -85,B 0,C 180,E1 -20640.119,E2 -20640.119} C_VEL
LIN {X 0,Y 217.787,Z 391.561,A -85,B 0,C 180,E1 -20641.836,E2 -20641.836} C_VEL
LIN {X 0,Y 216.715,Z 388.139,A -85,B 0,C 180,E1 -20642.438,E2 -20642.438} C_VEL
LIN {X 0,Y 215.865,Z 384.791,A -85,B 0,C 180,E1 -20642.953,E2 -20642.953} C_VEL
LIN {X 0,Y 216.262,Z 382.162,A -85,B 0,C 180,E1 -20645.803,E2 -20645.803} C_VEL
LIN {X 0,Y 216.02,Z 379.764,A -85,B 0,C 180,E1 -20648.663,E2 -20648.663} C_VEL
LIN {X 0,Y 215.411,Z 376.28,A -85,B 0,C 180,E1 -20653.25,E2 -20653.25} C_VEL
LIN {X 0,Y 215.007,Z 373.97,A -85,B 0,C 180,E1 -20656.65,E2 -20656.65} C_VEL
LIN {X 0,Y 214.531,Z 370.884,A -85,B 0,C 180,E1 -20661.838,E2 -20661.838} C_VEL
LIN {X 0,Y 214.163,Z 368.805,A -85,B 0,C 180,E1 -20666.089,E2 -20666.089} C_VEL
LIN {X 0,Y 213.825,Z 367.081,A -85,B 0,C 180,E1 -20670.459,E2 -20670.459} C_VEL
LIN {X 0,Y 213.836,Z 366.661,A -85,B 0,C 180,E1 -20672.603,E2 -20672.603} C_VEL
LIN {X 0,Y 213.862,Z 366.658,A -85,B 0,C 180,E1 -20676.952,E2 -20676.952} C_VEL
LIN {X 0,Y 213.953,Z 366.646,A -85,B 0,C 180,E1 -20682.803,E2 -20682.803} C_VEL
LIN {X 0,Y 213.96,Z 366.647,A -85,B 0,C 180,E1 -20686.705,E2 -20686.705} C_VEL
LIN {X 0,Y 214.145,Z 366.623,A -85,B 0,C 180,E1 -20690.554,E2 -20690.554} C_VEL
LIN {X 0,Y 214.095,Z 366.631,A -85,B 0,C 180,E1 -20694.347,E2 -20694.347} C_VEL
LIN {X 0,Y 214.449,Z 366.581,A -85,B 0,C 180,E1 -20698.12,E2 -20698.12} C_VEL
LIN {X 0,Y 214.554,Z 366.573,A -85,B 0,C 180,E1 -20699.998,E2 -20699.998} C_VEL
LIN {X 0,Y 214.451,Z 366.583,A -85,B 0,C 180,E1 -20701.876,E2 -20701.876} C_VEL
LIN {X 0,Y 214.148,Z 366.671,A -85,B 0,C 180,E1 -20703.762,E2 -20703.762} C_VEL
LIN {X 0,Y 214.402,Z 367.886,A -85,B 0,C 180,E1 -20707.532,E2 -20707.532} C_VEL
LIN {X 0,Y 214.45,Z 369.358,A -85,B 0,C 180,E1 -20711.338,E2 -20711.338} C_VEL
LIN {X 0,Y 214.48,Z 371.085,A -85,B 0,C 180,E1 -20715.195,E2 -20715.195} C_VEL
LIN {X 0,Y 214.436,Z 371.869,A -85,B 0,C 180,E1 -20716.847,E2 -20716.847} C_VEL
LIN {X 0,Y 215.468,Z 374.789,A -85,B 0,C 180,E1 -20717.4,E2 -20717.4} C_VEL
LIN {X 0,Y 216.696,Z 377.143,A -85,B 0,C 180,E1 -20717.956,E2 -20717.956} C_VEL
LIN {X 0,Y 220.293,Z 385.578,A -85,B 0,C 180,E1 -20719.83,E2 -20719.83} C_VEL
LIN {X 0,Y 222.773,Z 393.314,A -85,B 0,C 180,E1 -20721.513,E2 -20721.513} C_VEL
LIN {X 0,Y 224.668,Z 402.194,A -85,B 0,C 180,E1 -20723.504,E2 -20723.504} C_VEL
LIN {X 0,Y 225.612,Z 410.864,A -85,B 0,C 180,E1 -20725.59,E2 -20725.59} C_VEL
LIN {X 0,Y 225.55,Z 414.792,A -85,B 0,C 180,E1 -20726.608,E2 -20726.608} C_VEL
LIN {X 0,Y 223.389,Z 421.606,A -85,B 0,C 180,E1 -20728.245,E2 -20728.245} C_VEL
LIN {X 0,Y 221.316,Z 427.751,A -85,B 0,C 180,E1 -20730.077,E2 -20730.077} C_VEL
LIN {X 0,Y 218.876,Z 434.365,A -85,B 0,C 180,E1 -20732.552,E2 -20732.552} C_VEL
LIN {X 0,Y 216.794,Z 439.382,A -85,B 0,C 180,E1 -20735.057,E2 -20735.057} C_VEL
LIN {X 0,Y 215.449,Z 442.421,A -85,B 0,C 180,E1 -20737.004,E2 -20737.004} C_VEL
LIN {X 0,Y 213.978,Z 445.395,A -85,B 0,C 180,E1 -20739.629,E2 -20739.629} C_VEL
LIN {X 0,Y 213.233,Z 446.7,A -85,B 0,C 180,E1 -20741.235,E2 -20741.235} C_VEL
LIN {X 0,Y 212.279,Z 448.115,A -85,B 0,C 180,E1 -20744.044,E2 -20744.044} C_VEL
LIN {X 0,Y 211.647,Z 448.363,A -85,B 0,C 180,E1 -20746.928,E2 -20746.928} C_VEL
LIN {X 0,Y 211.376,Z 447.436,A -85,B 0,C 180,E1 -20749.878,E2 -20749.878} C_VEL
LIN {X 0,Y 211.528,Z 444.942,A -85,B 0,C 180,E1 -20753.267,E2 -20753.267} C_VEL
LIN {X 0,Y 211.97,Z 441.717,A -85,B 0,C 180,E1 -20755.98,E2 -20755.98} C_VEL
LIN {X 0,Y 212.631,Z 437.195,A -85,B 0,C 180,E1 -20758.676,E2 -20758.676} C_VEL
LIN {X 0,Y 213.368,Z 432.363,A -85,B 0,C 180,E1 -20760.914,E2 -20760.914} C_VEL
LIN {X 0,Y 214.431,Z 426.126,A -85,B 0,C 180,E1 -20763.212,E2 -20763.212} C_VEL
LIN {X 0,Y 215.206,Z 420.67,A -85,B 0,C 180,E1 -20764.876,E2 -20764.876} C_VEL
LIN {X 0,Y 216.495,Z 412.716,A -85,B 0,C 180,E1 -20766.855,E2 -20766.855} C_VEL
LIN {X 0,Y 217.631,Z 404.831,A -85,B 0,C 180,E1 -20768.446,E2 -20768.446} C_VEL
LIN {X 0,Y 217.931,Z 400.429,A -85,B 0,C 180,E1 -20769.22,E2 -20769.22} C_VEL
LIN {X 0,Y 216.78,Z 391.971,A -85,B 0,C 180,E1 -20770.588,E2 -20770.588} C_VEL
LIN {X 0,Y 215.425,Z 383.766,A -85,B 0,C 180,E1 -20771.697,E2 -20771.697} C_VEL
LIN {X 0,Y 213.623,Z 374.546,A -85,B 0,C 180,E1 -20772.713,E2 -20772.713} C_VEL
LIN {X 0,Y 212.523,Z 368.992,A -85,B 0,C 180,E1 -20773.272,E2 -20773.272} C_VEL
LIN {X 0,Y 212.854,Z 366.79,A -85,B 0,C 180,E1 -20776.391,E2 -20776.391} C_VEL
LIN {X 0,Y 213.659,Z 366.685,A -85,B 0,C 180,E1 -20780.667,E2 -20780.667} C_VEL
LIN {X 0,Y 213.936,Z 366.652,A -85,B 0,C 180,E1 -20782.447,E2 -20782.447} C_VEL
LIN {X 0,Y 214.434,Z 366.59,A -85,B 0,C 180,E1 -20788.119,E2 -20788.119} C_VEL
LIN {X 0,Y 214.542,Z 366.576,A -85,B 0,C 180,E1 -20789.998,E2 -20789.998} C_VEL
LIN {X 0,Y 214.438,Z 366.588,A -85,B 0,C 180,E1 -20791.876,E2 -20791.876} C_VEL
LIN {X 0,Y 214.239,Z 366.611,A -85,B 0,C 180,E1 -20797.537,E2 -20797.537} C_VEL
LIN {X 0,Y 214.038,Z 366.633,A -85,B 0,C 180,E1 -20801.36,E2 -20801.36} C_VEL
LIN {X 0,Y 213.923,Z 366.649,A -85,B 0,C 180,E1 -20805.235,E2 -20805.235} C_VEL
LIN {X 0,Y 213.829,Z 366.659,A -85,B 0,C 180,E1 -20809.186,E2 -20809.186} C_VEL
LIN {X 0,Y 213.836,Z 366.661,A -85,B 0,C 180,E1 -20813.225,E2 -20813.225} C_VEL
LIN {X 0,Y 213.817,Z 366.662,A -85,B 0,C 180,E1 -20817.449,E2 -20817.449} C_VEL
LIN {X 0,Y 213.767,Z 366.67,A -85,B 0,C 180,E1 -20821.734,E2 -20821.734} C_VEL
LIN {X 0,Y 213.747,Z 366.667,A -85,B 0,C 180,E1 -20826.284,E2 -20826.284} C_VEL
LIN {X 0,Y 213.817,Z 366.665,A -85,B 0,C 180,E1 -20831.097,E2 -20831.097} C_VEL
LIN {X 0,Y 213.824,Z 366.659,A -85,B 0,C 180,E1 -20833.692,E2 -20833.692} C_VEL
LIN {X 0,Y 213.828,Z 366.659,A -85,B 0,C 180,E1 -20836.356,E2 -20836.356} C_VEL
LIN {X 0,Y 213.811,Z 366.665,A -85,B 0,C 180,E1 -20839.11,E2 -20839.11} C_VEL
LIN {X 0,Y 213.744,Z 366.668,A -85,B 0,C 180,E1 -20843.715,E2 -20843.715} C_VEL
LIN {X 0,Y 213.783,Z 366.668,A -85,B 0,C 180,E1 -20848.725,E2 -20848.725} C_VEL
LIN {X 0,Y 213.814,Z 366.663,A -85,B 0,C 180,E1 -20852.604,E2 -20852.604} C_VEL
LIN {X 0,Y 213.858,Z 366.657,A -85,B 0,C 180,E1 -20856.942,E2 -20856.942} C_VEL
LIN {X 0,Y 213.929,Z 366.65,A -85,B 0,C 180,E1 -20862.299,E2 -20862.299} C_VEL
LIN {X 0,Y 213.97,Z 366.641,A -85,B 0,C 180,E1 -20866.71,E2 -20866.71} C_VEL
LIN {X 0,Y 214.185,Z 366.617,A -85,B 0,C 180,E1 -20870.559,E2 -20870.559} C_VEL
LIN {X 0,Y 214.237,Z 366.611,A -85,B 0,C 180,E1 -20872.462,E2 -20872.462} C_VEL
LIN {X 0,Y 214.436,Z 366.587,A -85,B 0,C 180,E1 -20878.124,E2 -20878.124} C_VEL
LIN {X 0,Y 214.54,Z 366.575,A -85,B 0,C 180,E1 -20880.002,E2 -20880.002} C_VEL
LIN {X 0,Y 214.438,Z 366.587,A -85,B 0,C 180,E1 -20881.88,E2 -20881.88} C_VEL
LIN {X 0,Y 214.239,Z 366.611,A -85,B 0,C 180,E1 -20887.542,E2 -20887.542} C_VEL
LIN {X 0,Y 214.034,Z 366.635,A -85,B 0,C 180,E1 -20891.364,E2 -20891.364} C_VEL
LIN {X 0,Y 213.926,Z 366.649,A -85,B 0,C 180,E1 -20895.239,E2 -20895.239} C_VEL
LIN {X 0,Y 213.861,Z 366.658,A -85,B 0,C 180,E1 -20899.187,E2 -20899.187} C_VEL
LIN {X 0,Y 213.841,Z 366.66,A -85,B 0,C 180,E1 -20903.229,E2 -20903.229} C_VEL
LIN {X 0,Y 213.823,Z 366.661,A -85,B 0,C 180,E1 -20907.452,E2 -20907.452} C_VEL
LIN {X 0,Y 213.771,Z 366.668,A -85,B 0,C 180,E1 -20911.739,E2 -20911.739} C_VEL
LIN {X 0,Y 213.739,Z 366.67,A -85,B 0,C 180,E1 -20916.291,E2 -20916.291} C_VEL
LIN {X 0,Y 213.708,Z 366.678,A -85,B 0,C 180,E1 -20921.128,E2 -20921.128} C_VEL
LIN {X 0,Y 213.888,Z 366.778,A -85,B 0,C 180,E1 -20926.79,E2 -20926.79} C_VEL
LIN {X 0,Y 214.773,Z 371.51,A -85,B 0,C 180,E1 -20931.755,E2 -20931.755} C_VEL
LIN {X 0,Y 215.285,Z 374.466,A -85,B 0,C 180,E1 -20934.701,E2 -20934.701} C_VEL
LIN {X 0,Y 215.004,Z 377.275,A -85,B 0,C 180,E1 -20937.365,E2 -20937.365} C_VEL
LIN {X 0,Y 213.875,Z 381.801,A -85,B 0,C 180,E1 -20941.548,E2 -20941.548} C_VEL
LIN {X 0,Y 212.81,Z 387.638,A -85,B 0,C 180,E1 -20946.768,E2 -20946.768} C_VEL
LIN {X 0,Y 214.221,Z 400.205,A -85,B 0,C 180,E1 -20947.873,E2 -20947.873} C_VEL
LIN {X 0,Y 214.972,Z 409.112,A -85,B 0,C 180,E1 -20948.926,E2 -20948.926} C_VEL
LIN {X 0,Y 215.338,Z 415.796,A -85,B 0,C 180,E1 -20949.865,E2 -20949.865} C_VEL
LIN {X 0,Y 214.813,Z 421.012,A -85,B 0,C 180,E1 -20950.677,E2 -20950.677} C_VEL
LIN {X 0,Y 213.231,Z 425.918,A -85,B 0,C 180,E1 -20951.504,E2 -20951.504} C_VEL
LIN {X 0,Y 209.065,Z 434.867,A -85,B 0,C 180,E1 -20953.35,E2 -20953.35} C_VEL
LIN {X 0,Y 207.946,Z 437.735,A -85,B 0,C 180,E1 -20954.059,E2 -20954.059} C_VEL
LIN {X 0,Y 207.241,Z 440.435,A -85,B 0,C 180,E1 -20954.819,E2 -20954.819} C_VEL
LIN {X 0,Y 206.16,Z 447.77,A -85,B 0,C 180,E1 -20957.201,E2 -20957.201} C_VEL
LIN {X 0,Y 205.237,Z 454.659,A -85,B 0,C 180,E1 -20960.144,E2 -20960.144} C_VEL
LIN {X 0,Y 204.731,Z 459.841,A -85,B 0,C 180,E1 -20963.102,E2 -20963.102} C_VEL
LIN {X 0,Y 204.571,Z 462.48,A -85,B 0,C 180,E1 -20965.077,E2 -20965.077} C_VEL
LIN {X 0,Y 204.657,Z 465.342,A -85,B 0,C 180,E1 -20968.035,E2 -20968.035} C_VEL
LIN {X 0,Y 204.676,Z 466.54,A -85,B 0,C 180,E1 -20970.003,E2 -20970.003} C_VEL
LIN {X 0,Y 204.56,Z 467.245,A -85,B 0,C 180,E1 -20971.971,E2 -20971.971} C_VEL
LIN {X 0,Y 204.439,Z 467.375,A -85,B 0,C 180,E1 -20974.472,E2 -20974.472} C_VEL
LIN {X 0,Y 204.76,Z 466.222,A -85,B 0,C 180,E1 -20977.894,E2 -20977.894} C_VEL
LIN {X 0,Y 205.213,Z 464.922,A -85,B 0,C 180,E1 -20979.862,E2 -20979.862} C_VEL
LIN {X 0,Y 206.348,Z 461.965,A -85,B 0,C 180,E1 -20982.793,E2 -20982.793} C_VEL
LIN {X 0,Y 207.987,Z 457.787,A -85,B 0,C 180,E1 -20985.686,E2 -20985.686} C_VEL
LIN {X 0,Y 210.246,Z 452.222,A -85,B 0,C 180,E1 -20988.518,E2 -20988.518} C_VEL
LIN {X 0,Y 212.644,Z 446.199,A -85,B 0,C 180,E1 -20990.814,E2 -20990.814} C_VEL
LIN {X 0,Y 214.476,Z 440.41,A -85,B 0,C 180,E1 -20992.648,E2 -20992.648} C_VEL
LIN {X 0,Y 215.75,Z 433.178,A -85,B 0,C 180,E1 -20994.651,E2 -20994.651} C_VEL
LIN {X 0,Y 216.33,Z 425.479,A -85,B 0,C 180,E1 -20996.535,E2 -20996.535} C_VEL
LIN {X 0,Y 216.314,Z 418.016,A -85,B 0,C 180,E1 -20998.175,E2 -20998.175} C_VEL
LIN {X 0,Y 215.442,Z 409.202,A -85,B 0,C 180,E1 -20999.971,E2 -20999.971} C_VEL
LIN {X 0,Y 213.76,Z 400.058,A -85,B 0,C 180,E1 -21001.741,E2 -21001.741} C_VEL
LIN {X 0,Y 211.537,Z 391.794,A -85,B 0,C 180,E1 -21003.299,E2 -21003.299} C_VEL
LIN {X 0,Y 210.455,Z 388.371,A -85,B 0,C 180,E1 -21003.944,E2 -21003.944} C_VEL
LIN {X 0,Y 209.268,Z 385.28,A -85,B 0,C 180,E1 -21004.547,E2 -21004.547} C_VEL
LIN {X 0,Y 209.118,Z 384.356,A -85,B 0,C 180,E1 -21004.702,E2 -21004.702} C_VEL
LIN {X 0,Y 209.195,Z 382.224,A -85,B 0,C 180,E1 -21007.211,E2 -21007.211} C_VEL
LIN {X 0,Y 208.899,Z 380.25,A -85,B 0,C 180,E1 -21009.736,E2 -21009.736} C_VEL
LIN {X 0,Y 208.565,Z 378.327,A -85,B 0,C 180,E1 -21012.375,E2 -21012.375} C_VEL
LIN {X 0,Y 208.219,Z 376.443,A -85,B 0,C 180,E1 -21015.141,E2 -21015.141} C_VEL
LIN {X 0,Y 207.71,Z 373.512,A -85,B 0,C 180,E1 -21019.991,E2 -21019.991} C_VEL
LIN {X 0,Y 207.393,Z 371.227,A -85,B 0,C 180,E1 -21024.423,E2 -21024.423} C_VEL
LIN {X 0,Y 207.023,Z 369.165,A -85,B 0,C 180,E1 -21029.386,E2 -21029.386} C_VEL
LIN {X 0,Y 206.798,Z 367.77,A -85,B 0,C 180,E1 -21033.779,E2 -21033.779} C_VEL
LIN {X 0,Y 206.767,Z 367.541,A -85,B 0,C 180,E1 -21038.043,E2 -21038.043} C_VEL
LIN {X 0,Y 206.883,Z 367.529,A -85,B 0,C 180,E1 -21042.196,E2 -21042.196} C_VEL
LIN {X 0,Y 206.903,Z 367.525,A -85,B 0,C 180,E1 -21046.243,E2 -21046.243} C_VEL
LIN {X 0,Y 207.089,Z 367.502,A -85,B 0,C 180,E1 -21050.229,E2 -21050.229} C_VEL
LIN {X 0,Y 207.057,Z 367.506,A -85,B 0,C 180,E1 -21054.154,E2 -21054.154} C_VEL
LIN {X 0,Y 207.385,Z 367.461,A -85,B 0,C 180,E1 -21058.056,E2 -21058.056} C_VEL
LIN {X 0,Y 207.519,Z 367.449,A -85,B 0,C 180,E1 -21059.998,E2 -21059.998} C_VEL
LIN {X 0,Y 207.413,Z 367.686,A -85,B 0,C 180,E1 -21061.94,E2 -21061.94} C_VEL
LIN {X 0,Y 207.453,Z 369.477,A -85,B 0,C 180,E1 -21067.786,E2 -21067.786} C_VEL
LIN {X 0,Y 207.493,Z 370.968,A -85,B 0,C 180,E1 -21071.724,E2 -21071.724} C_VEL
LIN {X 0,Y 207.538,Z 372.491,A -85,B 0,C 180,E1 -21075.024,E2 -21075.024} C_VEL
LIN {X 0,Y 208.614,Z 375.324,A -85,B 0,C 180,E1 -21075.633,E2 -21075.633} C_VEL
LIN {X 0,Y 209.957,Z 377.619,A -85,B 0,C 180,E1 -21076.278,E2 -21076.278} C_VEL
LIN {X 0,Y 213.568,Z 385.802,A -85,B 0,C 180,E1 -21078.265,E2 -21078.265} C_VEL
LIN {X 0,Y 216.004,Z 392.949,A -85,B 0,C 180,E1 -21079.974,E2 -21079.974} C_VEL
LIN {X 0,Y 217.886,Z 400.728,A -85,B 0,C 180,E1 -21081.845,E2 -21081.845} C_VEL
LIN {X 0,Y 218.897,Z 407.705,A -85,B 0,C 180,E1 -21083.581,E2 -21083.581} C_VEL
LIN {X 0,Y 219.279,Z 413.304,A -85,B 0,C 180,E1 -21085.061,E2 -21085.061} C_VEL
LIN {X 0,Y 218.979,Z 416.89,A -85,B 0,C 180,E1 -21086.015,E2 -21086.015} C_VEL
LIN {X 0,Y 216.311,Z 424.664,A -85,B 0,C 180,E1 -21088.055,E2 -21088.055} C_VEL
LIN {X 0,Y 213.958,Z 430.932,A -85,B 0,C 180,E1 -21090.183,E2 -21090.183} C_VEL
LIN {X 0,Y 211.461,Z 436.866,A -85,B 0,C 180,E1 -21092.771,E2 -21092.771} C_VEL
LIN {X 0,Y 209.397,Z 441.462,A -85,B 0,C 180,E1 -21095.422,E2 -21095.422} C_VEL
LIN {X 0,Y 207.309,Z 445.549,A -85,B 0,C 180,E1 -21098.761,E2 -21098.761} C_VEL
LIN {X 0,Y 206.064,Z 447.509,A -85,B 0,C 180,E1 -21101.378,E2 -21101.378} C_VEL
LIN {X 0,Y 205.181,Z 448.545,A -85,B 0,C 180,E1 -21104,E2 -21104} C_VEL
LIN {X 0,Y 204.598,Z 448.704,A -85,B 0,C 180,E1 -21106.603,E2 -21106.603} C_VEL
LIN {X 0,Y 204.325,Z 448.009,A -85,B 0,C 180,E1 -21109.189,E2 -21109.189} C_VEL
LIN {X 0,Y 204.313,Z 446.008,A -85,B 0,C 180,E1 -21112.29,E2 -21112.29} C_VEL
LIN {X 0,Y 204.757,Z 442.651,A -85,B 0,C 180,E1 -21115.459,E2 -21115.459} C_VEL
LIN {X 0,Y 205.528,Z 437.509,A -85,B 0,C 180,E1 -21118.741,E2 -21118.741} C_VEL
LIN {X 0,Y 206.259,Z 432.925,A -85,B 0,C 180,E1 -21120.949,E2 -21120.949} C_VEL
LIN {X 0,Y 207.326,Z 426.783,A -85,B 0,C 180,E1 -21123.308,E2 -21123.308} C_VEL
LIN {X 0,Y 208.248,Z 420.663,A -85,B 0,C 180,E1 -21125.231,E2 -21125.231} C_VEL
LIN {X 0,Y 209.43,Z 413.661,A -85,B 0,C 180,E1 -21127.036,E2 -21127.036} C_VEL
LIN {X 0,Y 210.523,Z 406.102,A -85,B 0,C 180,E1 -21128.642,E2 -21128.642} C_VEL
LIN {X 0,Y 211.006,Z 401.704,A -85,B 0,C 180,E1 -21129.463,E2 -21129.463} C_VEL
LIN {X 0,Y 209.843,Z 393.041,A -85,B 0,C 180,E1 -21130.938,E2 -21130.938} C_VEL
LIN {X 0,Y 208.468,Z 384.537,A -85,B 0,C 180,E1 -21132.145,E2 -21132.145} C_VEL
LIN {X 0,Y 206.612,Z 374.914,A -85,B 0,C 180,E1 -21133.253,E2 -21133.253} C_VEL
LIN {X 0,Y 205.512,Z 369.31,A -85,B 0,C 180,E1 -21133.821,E2 -21133.821} C_VEL
LIN {X 0,Y 205.745,Z 367.677,A -85,B 0,C 180,E1 -21136.163,E2 -21136.163} C_VEL
LIN {X 0,Y 206.588,Z 367.566,A -85,B 0,C 180,E1 -21140.581,E2 -21140.581} C_VEL
LIN {X 0,Y 206.959,Z 367.521,A -85,B 0,C 180,E1 -21144.15,E2 -21144.15} C_VEL
LIN {X 0,Y 207.369,Z 367.47,A -85,B 0,C 180,E1 -21148.055,E2 -21148.055} C_VEL
LIN {X 0,Y 207.506,Z 367.452,A -85,B 0,C 180,E1 -21149.998,E2 -21149.998} C_VEL
LIN {X 0,Y 207.375,Z 367.468,A -85,B 0,C 180,E1 -21151.94,E2 -21151.94} C_VEL
LIN {X 0,Y 207.18,Z 367.491,A -85,B 0,C 180,E1 -21157.796,E2 -21157.796} C_VEL
LIN {X 0,Y 206.973,Z 367.514,A -85,B 0,C 180,E1 -21161.753,E2 -21161.753} C_VEL
LIN {X 0,Y 206.857,Z 367.532,A -85,B 0,C 180,E1 -21165.769,E2 -21165.769} C_VEL
LIN {X 0,Y 206.773,Z 367.538,A -85,B 0,C 180,E1 -21169.867,E2 -21169.867} C_VEL
LIN {X 0,Y 206.752,Z 367.543,A -85,B 0,C 180,E1 -21174.071,E2 -21174.071} C_VEL
LIN {X 0,Y 206.732,Z 367.541,A -85,B 0,C 180,E1 -21178.417,E2 -21178.417} C_VEL
LIN {X 0,Y 206.697,Z 367.55,A -85,B 0,C 180,E1 -21182.955,E2 -21182.955} C_VEL
LIN {X 0,Y 206.733,Z 367.544,A -85,B 0,C 180,E1 -21187.725,E2 -21187.725} C_VEL
LIN {X 0,Y 206.741,Z 367.544,A -85,B 0,C 180,E1 -21191.597,E2 -21191.597} C_VEL
LIN {X 0,Y 206.733,Z 367.543,A -85,B 0,C 180,E1 -21195.549,E2 -21195.549} C_VEL
LIN {X 0,Y 206.731,Z 367.544,A -85,B 0,C 180,E1 -21199.768,E2 -21199.768} C_VEL
LIN {X 0,Y 206.719,Z 367.546,A -85,B 0,C 180,E1 -21204.695,E2 -21204.695} C_VEL
LIN {X 0,Y 206.711,Z 367.546,A -85,B 0,C 180,E1 -21209.34,E2 -21209.34} C_VEL
LIN {X 0,Y 206.726,Z 367.545,A -85,B 0,C 180,E1 -21213.774,E2 -21213.774} C_VEL
LIN {X 0,Y 206.78,Z 367.539,A -85,B 0,C 180,E1 -21218.048,E2 -21218.048} C_VEL
LIN {X 0,Y 206.874,Z 367.528,A -85,B 0,C 180,E1 -21222.199,E2 -21222.199} C_VEL
LIN {X 0,Y 206.904,Z 367.524,A -85,B 0,C 180,E1 -21226.247,E2 -21226.247} C_VEL
LIN {X 0,Y 207.122,Z 367.498,A -85,B 0,C 180,E1 -21230.234,E2 -21230.234} C_VEL
LIN {X 0,Y 207.178,Z 367.492,A -85,B 0,C 180,E1 -21232.203,E2 -21232.203} C_VEL
LIN {X 0,Y 207.373,Z 367.466,A -85,B 0,C 180,E1 -21238.06,E2 -21238.06} C_VEL
LIN {X 0,Y 207.505,Z 367.451,A -85,B 0,C 180,E1 -21240.002,E2 -21240.002} C_VEL
LIN {X 0,Y 207.374,Z 367.466,A -85,B 0,C 180,E1 -21241.944,E2 -21241.944} C_VEL
LIN {X 0,Y 207.18,Z 367.492,A -85,B 0,C 180,E1 -21247.8,E2 -21247.8} C_VEL
LIN {X 0,Y 206.967,Z 367.514,A -85,B 0,C 180,E1 -21251.758,E2 -21251.758} C_VEL
LIN {X 0,Y 206.86,Z 367.531,A -85,B 0,C 180,E1 -21255.773,E2 -21255.773} C_VEL
LIN {X 0,Y 206.792,Z 367.535,A -85,B 0,C 180,E1 -21259.87,E2 -21259.87} C_VEL
LIN {X 0,Y 206.757,Z 367.542,A -85,B 0,C 180,E1 -21264.075,E2 -21264.075} C_VEL
LIN {X 0,Y 206.738,Z 367.541,A -85,B 0,C 180,E1 -21268.421,E2 -21268.421} C_VEL
LIN {X 0,Y 206.697,Z 367.551,A -85,B 0,C 180,E1 -21272.96,E2 -21272.96} C_VEL
LIN {X 0,Y 206.674,Z 367.549,A -85,B 0,C 180,E1 -21277.743,E2 -21277.743} C_VEL
LIN {X 0,Y 206.639,Z 367.557,A -85,B 0,C 180,E1 -21281.566,E2 -21281.566} C_VEL
LIN {X 0,Y 206.823,Z 367.602,A -85,B 0,C 180,E1 -21286.599,E2 -21286.599} C_VEL
LIN {X 0,Y 207.586,Z 371.777,A -85,B 0,C 180,E1 -21291.142,E2 -21291.142} C_VEL
LIN {X 0,Y 208.191,Z 374.624,A -85,B 0,C 180,E1 -21294.116,E2 -21294.116} C_VEL
LIN {X 0,Y 208.165,Z 376.661,A -85,B 0,C 180,E1 -21296.15,E2 -21296.15} C_VEL
LIN {X 0,Y 207.328,Z 380.081,A -85,B 0,C 180,E1 -21299.441,E2 -21299.441} C_VEL
LIN {X 0,Y 206.04,Z 385.726,A -85,B 0,C 180,E1 -21304.765,E2 -21304.765} C_VEL
LIN {X 0,Y 205.805,Z 387.23,A -85,B 0,C 180,E1 -21306.183,E2 -21306.183} C_VEL
LIN {X 0,Y 207.113,Z 399.087,A -85,B 0,C 180,E1 -21307.265,E2 -21307.265} C_VEL
LIN {X 0,Y 207.903,Z 408.67,A -85,B 0,C 180,E1 -21308.434,E2 -21308.434} C_VEL
LIN {X 0,Y 208.394,Z 417.558,A -85,B 0,C 180,E1 -21309.78,E2 -21309.78} C_VEL
LIN {X 0,Y 208.676,Z 425.331,A -85,B 0,C 180,E1 -21311.205,E2 -21311.205} C_VEL
LIN {X 0,Y 208.639,Z 431.859,A -85,B 0,C 180,E1 -21312.608,E2 -21312.608} C_VEL
LIN {X 0,Y 207.531,Z 438.555,A -85,B 0,C 180,E1 -21314.284,E2 -21314.284} C_VEL
LIN {X 0,Y 207.241,Z 440.435,A -85,B 0,C 180,E1 -21314.819,E2 -21314.819} C_VEL
LIN {X 0,Y 205.965,Z 444.367,A -85,B 0,C 180,E1 -21316.002,E2 -21316.002} C_VEL
LIN {X 0,Y 203.848,Z 447.876,A -85,B 0,C 180,E1 -21317.215,E2 -21317.215} C_VEL
LIN {X 0,Y 199.297,Z 453.957,A -85,B 0,C 180,E1 -21319.847,E2 -21319.847} C_VEL
LIN {X 0,Y 197.95,Z 456.673,A -85,B 0,C 180,E1 -21321.308,E2 -21321.308} C_VEL
LIN {X 0,Y 197.784,Z 457.553,A -85,B 0,C 180,E1 -21321.811,E2 -21321.811} C_VEL
LIN {X 0,Y 197.581,Z 460.625,A -85,B 0,C 180,E1 -21323.877,E2 -21323.877} C_VEL
LIN {X 0,Y 197.469,Z 462.987,A -85,B 0,C 180,E1 -21325.921,E2 -21325.921} C_VEL
LIN {X 0,Y 197.567,Z 464.798,A -85,B 0,C 180,E1 -21327.964,E2 -21327.964} C_VEL
LIN {X 0,Y 197.61,Z 466.08,A -85,B 0,C 180,E1 -21330.003,E2 -21330.003} C_VEL
LIN {X 0,Y 197.471,Z 466.863,A -85,B 0,C 180,E1 -21332.042,E2 -21332.042} C_VEL
LIN {X 0,Y 197.348,Z 467.098,A -85,B 0,C 180,E1 -21334.317,E2 -21334.317} C_VEL
LIN {X 0,Y 197.714,Z 466.018,A -85,B 0,C 180,E1 -21338.177,E2 -21338.177} C_VEL
LIN {X 0,Y 198.211,Z 464.81,A -85,B 0,C 180,E1 -21340.214,E2 -21340.214} C_VEL
LIN {X 0,Y 199.418,Z 461.948,A -85,B 0,C 180,E1 -21343.245,E2 -21343.245} C_VEL
LIN {X 0,Y 201.147,Z 457.87,A -85,B 0,C 180,E1 -21346.234,E2 -21346.234} C_VEL
LIN {X 0,Y 203.547,Z 452.453,A -85,B 0,C 180,E1 -21349.151,E2 -21349.151} C_VEL
LIN {X 0,Y 206.529,Z 445.285,A -85,B 0,C 180,E1 -21351.985,E2 -21351.985} C_VEL
LIN {X 0,Y 208.304,Z 439.449,A -85,B 0,C 180,E1 -21353.885,E2 -21353.885} C_VEL
LIN {X 0,Y 209.523,Z 432.56,A -85,B 0,C 180,E1 -21355.855,E2 -21355.855} C_VEL
LIN {X 0,Y 210.103,Z 424.37,A -85,B 0,C 180,E1 -21357.927,E2 -21357.927} C_VEL
LIN {X 0,Y 209.911,Z 416.341,A -85,B 0,C 180,E1 -21359.784,E2 -21359.784} C_VEL
LIN {X 0,Y 209.125,Z 408.597,A -85,B 0,C 180,E1 -21361.46,E2 -21361.46} C_VEL
LIN {X 0,Y 207.709,Z 400.483,A -85,B 0,C 180,E1 -21363.126,E2 -21363.126} C_VEL
LIN {X 0,Y 205.359,Z 392.191,A -85,B 0,C 180,E1 -21364.871,E2 -21364.871} C_VEL
LIN {X 0,Y 203.926,Z 388.369,A -85,B 0,C 180,E1 -21365.731,E2 -21365.731} C_VEL
LIN {X 0,Y 202.516,Z 385.074,A -85,B 0,C 180,E1 -21366.507,E2 -21366.507} C_VEL
LIN {X 0,Y 202.234,Z 383.86,A -85,B 0,C 180,E1 -21366.751,E2 -21366.751} C_VEL
LIN {X 0,Y 201.875,Z 381.394,A -85,B 0,C 180,E1 -21370.011,E2 -21370.011} C_VEL
LIN {X 0,Y 201.347,Z 378.465,A -85,B 0,C 180,E1 -21374.278,E2 -21374.278} C_VEL
LIN {X 0,Y 200.943,Z 375.984,A -85,B 0,C 180,E1 -21378.352,E2 -21378.352} C_VEL
LIN {X 0,Y 200.536,Z 373.336,A -85,B 0,C 180,E1 -21383.43,E2 -21383.43} C_VEL
LIN {X 0,Y 200.192,Z 371.303,A -85,B 0,C 180,E1 -21388.222,E2 -21388.222} C_VEL
LIN {X 0,Y 199.957,Z 369.783,A -85,B 0,C 180,E1 -21392.81,E2 -21392.81} C_VEL
LIN {X 0,Y 199.764,Z 368.711,A -85,B 0,C 180,E1 -21397.23,E2 -21397.23} C_VEL
LIN {X 0,Y 199.806,Z 368.408,A -85,B 0,C 180,E1 -21401.757,E2 -21401.757} C_VEL
LIN {X 0,Y 199.844,Z 368.404,A -85,B 0,C 180,E1 -21405.747,E2 -21405.747} C_VEL
LIN {X 0,Y 200.032,Z 368.382,A -85,B 0,C 180,E1 -21409.88,E2 -21409.88} C_VEL
LIN {X 0,Y 200.02,Z 368.382,A -85,B 0,C 180,E1 -21413.947,E2 -21413.947} C_VEL
LIN {X 0,Y 200.349,Z 368.464,A -85,B 0,C 180,E1 -21417.988,E2 -21417.988} C_VEL
LIN {X 0,Y 200.563,Z 368.821,A -85,B 0,C 180,E1 -21419.998,E2 -21419.998} C_VEL
LIN {X 0,Y 200.322,Z 369.88,A -85,B 0,C 180,E1 -21424.022,E2 -21424.022} C_VEL
LIN {X 0,Y 200.52,Z 371.086,A -85,B 0,C 180,E1 -21428.057,E2 -21428.057} C_VEL
LIN {X 0,Y 200.532,Z 372.577,A -85,B 0,C 180,E1 -21432.137,E2 -21432.137} C_VEL
LIN {X 0,Y 200.526,Z 372.932,A -85,B 0,C 180,E1 -21432.908,E2 -21432.908} C_VEL
LIN {X 0,Y 201.673,Z 375.824,A -85,B 0,C 180,E1 -21433.603,E2 -21433.603} C_VEL
LIN {X 0,Y 203.232,Z 378.13,A -85,B 0,C 180,E1 -21434.378,E2 -21434.378} C_VEL
LIN {X 0,Y 205.799,Z 383.556,A -85,B 0,C 180,E1 -21435.852,E2 -21435.852} C_VEL
LIN {X 0,Y 209.105,Z 391.974,A -85,B 0,C 180,E1 -21438.111,E2 -21438.111} C_VEL
LIN {X 0,Y 211.114,Z 399.054,A -85,B 0,C 180,E1 -21439.949,E2 -21439.949} C_VEL
LIN {X 0,Y 212.441,Z 407.284,A -85,B 0,C 180,E1 -21442.13,E2 -21442.13} C_VEL
LIN {X 0,Y 212.938,Z 413.465,A -85,B 0,C 180,E1 -21443.846,E2 -21443.846} C_VEL
LIN {X 0,Y 212.71,Z 418.131,A -85,B 0,C 180,E1 -21445.173,E2 -21445.173} C_VEL
LIN {X 0,Y 210.027,Z 425.479,A -85,B 0,C 180,E1 -21447.205,E2 -21447.205} C_VEL
LIN {X 0,Y 207.693,Z 431.307,A -85,B 0,C 180,E1 -21449.248,E2 -21449.248} C_VEL
LIN {X 0,Y 205.026,Z 437.17,A -85,B 0,C 180,E1 -21451.874,E2 -21451.874} C_VEL
LIN {X 0,Y 203.293,Z 440.766,A -85,B 0,C 180,E1 -21453.928,E2 -21453.928} C_VEL
LIN {X 0,Y 201.4,Z 444.336,A -85,B 0,C 180,E1 -21456.617,E2 -21456.617} C_VEL
LIN {X 0,Y 199.858,Z 446.851,A -85,B 0,C 180,E1 -21459.316,E2 -21459.316} C_VEL
LIN {X 0,Y 198.655,Z 448.486,A -85,B 0,C 180,E1 -21462.232,E2 -21462.232} C_VEL
LIN {X 0,Y 197.768,Z 449.106,A -85,B 0,C 180,E1 -21465.291,E2 -21465.291} C_VEL
LIN {X 0,Y 197.267,Z 448.571,A -85,B 0,C 180,E1 -21468.428,E2 -21468.428} C_VEL
LIN {X 0,Y 197.178,Z 446.727,A -85,B 0,C 180,E1 -21471.638,E2 -21471.638} C_VEL
LIN {X 0,Y 197.552,Z 443.549,A -85,B 0,C 180,E1 -21474.904,E2 -21474.904} C_VEL
LIN {X 0,Y 198.281,Z 438.772,A -85,B 0,C 180,E1 -21478.28,E2 -21478.28} C_VEL
LIN {X 0,Y 199.197,Z 433.148,A -85,B 0,C 180,E1 -21481.126,E2 -21481.126} C_VEL
LIN {X 0,Y 200.224,Z 427.437,A -85,B 0,C 180,E1 -21483.412,E2 -21483.412} C_VEL
LIN {X 0,Y 201.127,Z 421.743,A -85,B 0,C 180,E1 -21485.295,E2 -21485.295} C_VEL
LIN {X 0,Y 202.394,Z 414.43,A -85,B 0,C 180,E1 -21487.272,E2 -21487.272} C_VEL
LIN {X 0,Y 203.443,Z 407.342,A -85,B 0,C 180,E1 -21488.856,E2 -21488.856} C_VEL
LIN {X 0,Y 204.02,Z 402.277,A -85,B 0,C 180,E1 -21489.848,E2 -21489.848} C_VEL
LIN {X 0,Y 202.678,Z 392.479,A -85,B 0,C 180,E1 -21491.564,E2 -21491.564} C_VEL
LIN {X 0,Y 201.382,Z 384.303,A -85,B 0,C 180,E1 -21492.741,E2 -21492.741} C_VEL
LIN {X 0,Y 199.582,Z 375.07,A -85,B 0,C 180,E1 -21493.832,E2 -21493.832} C_VEL
LIN {X 0,Y 198.5,Z 369.631,A -85,B 0,C 180,E1 -21494.401,E2 -21494.401} C_VEL
LIN {X 0,Y 198.718,Z 368.551,A -85,B 0,C 180,E1 -21496.186,E2 -21496.186} C_VEL
LIN {X 0,Y 199.525,Z 368.446,A -85,B 0,C 180,E1 -21500.477,E2 -21500.477} C_VEL
LIN {X 0,Y 199.904,Z 368.399,A -85,B 0,C 180,E1 -21503.943,E2 -21503.943} C_VEL
LIN {X 0,Y 200.307,Z 368.349,A -85,B 0,C 180,E1 -21507.987,E2 -21507.987} C_VEL
LIN {X 0,Y 200.471,Z 368.328,A -85,B 0,C 180,E1 -21509.997,E2 -21509.997} C_VEL
LIN {X 0,Y 200.027,Z 368.383,A -85,B 0,C 180,E1 -21514.027,E2 -21514.027} C_VEL
LIN {X 0,Y 200.123,Z 368.37,A -85,B 0,C 180,E1 -21518.073,E2 -21518.073} C_VEL
LIN {X 0,Y 199.905,Z 368.394,A -85,B 0,C 180,E1 -21522.175,E2 -21522.175} C_VEL
LIN {X 0,Y 199.794,Z 368.409,A -85,B 0,C 180,E1 -21526.341,E2 -21526.341} C_VEL
LIN {X 0,Y 199.689,Z 368.419,A -85,B 0,C 180,E1 -21530.603,E2 -21530.603} C_VEL
LIN {X 0,Y 199.662,Z 368.426,A -85,B 0,C 180,E1 -21534.983,E2 -21534.983} C_VEL
LIN {X 0,Y 199.663,Z 368.426,A -85,B 0,C 180,E1 -21539.521,E2 -21539.521} C_VEL
LIN {X 0,Y 199.652,Z 368.426,A -85,B 0,C 180,E1 -21542.351,E2 -21542.351} C_VEL
LIN {X 0,Y 199.651,Z 368.424,A -85,B 0,C 180,E1 -21546.753,E2 -21546.753} C_VEL
LIN {X 0,Y 199.712,Z 368.422,A -85,B 0,C 180,E1 -21549.3,E2 -21549.3} C_VEL
LIN {X 0,Y 199.69,Z 368.421,A -85,B 0,C 180,E1 -21552.35,E2 -21552.35} C_VEL
LIN {X 0,Y 199.682,Z 368.422,A -85,B 0,C 180,E1 -21555.261,E2 -21555.261} C_VEL
LIN {X 0,Y 199.685,Z 368.422,A -85,B 0,C 180,E1 -21558.036,E2 -21558.036} C_VEL
LIN {X 0,Y 199.69,Z 368.424,A -85,B 0,C 180,E1 -21560.735,E2 -21560.735} C_VEL
LIN {X 0,Y 199.622,Z 368.43,A -85,B 0,C 180,E1 -21565.718,E2 -21565.718} C_VEL
LIN {X 0,Y 199.691,Z 368.422,A -85,B 0,C 180,E1 -21568.138,E2 -21568.138} C_VEL
LIN {X 0,Y 199.677,Z 368.425,A -85,B 0,C 180,E1 -21572.773,E2 -21572.773} C_VEL
LIN {X 0,Y 199.747,Z 368.414,A -85,B 0,C 180,E1 -21577.233,E2 -21577.233} C_VEL
LIN {X 0,Y 199.827,Z 368.404,A -85,B 0,C 180,E1 -21581.723,E2 -21581.723} C_VEL
LIN {X 0,Y 199.84,Z 368.403,A -85,B 0,C 180,E1 -21585.751,E2 -21585.751} C_VEL
LIN {X 0,Y 200.065,Z 368.375,A -85,B 0,C 180,E1 -21589.886,E2 -21589.886} C_VEL
LIN {X 0,Y 200.121,Z 368.37,A -85,B 0,C 180,E1 -21591.927,E2 -21591.927} C_VEL
LIN {X 0,Y 200.313,Z 368.345,A -85,B 0,C 180,E1 -21597.991,E2 -21597.991} C_VEL
LIN {X 0,Y 200.47,Z 368.328,A -85,B 0,C 180,E1 -21600.002,E2 -21600.002} C_VEL
LIN {X 0,Y 200.025,Z 368.378,A -85,B 0,C 180,E1 -21604.032,E2 -21604.032} C_VEL
LIN {X 0,Y 200.123,Z 368.369,A -85,B 0,C 180,E1 -21608.077,E2 -21608.077} C_VEL
LIN {X 0,Y 199.898,Z 368.392,A -85,B 0,C 180,E1 -21612.18,E2 -21612.18} C_VEL
LIN {X 0,Y 199.798,Z 368.408,A -85,B 0,C 180,E1 -21616.346,E2 -21616.346} C_VEL
LIN {X 0,Y 199.817,Z 368.405,A -85,B 0,C 180,E1 -21618.456,E2 -21618.456} C_VEL
LIN {X 0,Y 199.73,Z 368.418,A -85,B 0,C 180,E1 -21623.82,E2 -21623.82} C_VEL
LIN {X 0,Y 199.707,Z 368.417,A -85,B 0,C 180,E1 -21628.389,E2 -21628.389} C_VEL
LIN {X 0,Y 199.672,Z 368.424,A -85,B 0,C 180,E1 -21632.361,E2 -21632.361} C_VEL
LIN {X 0,Y 199.618,Z 368.43,A -85,B 0,C 180,E1 -21636.766,E2 -21636.766} C_VEL
LIN {X 0,Y 199.604,Z 368.433,A -85,B 0,C 180,E1 -21639.331,E2 -21639.331} C_VEL
LIN {X 0,Y 199.62,Z 368.431,A -85,B 0,C 180,E1 -21644.762,E2 -21644.762} C_VEL
LIN {X 0,Y 199.798,Z 368.616,A -85,B 0,C 180,E1 -21646.64,E2 -21646.64} C_VEL
LIN {X 0,Y 200.766,Z 373.609,A -85,B 0,C 180,E1 -21652.226,E2 -21652.226} C_VEL
LIN {X 0,Y 201.124,Z 376.023,A -85,B 0,C 180,E1 -21654.794,E2 -21654.794} C_VEL
LIN {X 0,Y 200.883,Z 378.29,A -85,B 0,C 180,E1 -21657.106,E2 -21657.106} C_VEL
LIN {X 0,Y 199.619,Z 382.898,A -85,B 0,C 180,E1 -21661.666,E2 -21661.666} C_VEL
LIN {X 0,Y 198.793,Z 387.116,A -85,B 0,C 180,E1 -21665.624,E2 -21665.624} C_VEL
LIN {X 0,Y 200.165,Z 399.308,A -85,B 0,C 180,E1 -21666.779,E2 -21666.779} C_VEL
LIN {X 0,Y 200.881,Z 408.238,A -85,B 0,C 180,E1 -21667.911,E2 -21667.911} C_VEL
LIN {X 0,Y 201.389,Z 417.156,A -85,B 0,C 180,E1 -21669.311,E2 -21669.311} C_VEL
LIN {X 0,Y 201.639,Z 425.868,A -85,B 0,C 180,E1 -21670.983,E2 -21670.983} C_VEL
LIN {X 0,Y 201.516,Z 432.511,A -85,B 0,C 180,E1 -21672.497,E2 -21672.497} C_VEL
LIN {X 0,Y 200.216,Z 440.198,A -85,B 0,C 180,E1 -21674.571,E2 -21674.571} C_VEL
LIN {X 0,Y 199.011,Z 448.094,A -85,B 0,C 180,E1 -21677.252,E2 -21677.252} C_VEL
LIN {X 0,Y 198.22,Z 453.831,A -85,B 0,C 180,E1 -21679.791,E2 -21679.791} C_VEL
LIN {X 0,Y 197.784,Z 457.553,A -85,B 0,C 180,E1 -21681.811,E2 -21681.811} C_VEL
LIN {X 0,Y 196.967,Z 460.031,A -85,B 0,C 180,E1 -21683.349,E2 -21683.349} C_VEL
LIN {X 0,Y 195.36,Z 461.996,A -85,B 0,C 180,E1 -21684.917,E2 -21684.917} C_VEL
LIN {X 0,Y 191.706,Z 464.683,A -85,B 0,C 180,E1 -21688.208,E2 -21688.208} C_VEL
LIN {X 0,Y 190.478,Z 465.826,A -85,B 0,C 180,E1 -21690.553,E2 -21690.553} C_VEL
LIN {X 0,Y 190.384,Z 466.452,A -85,B 0,C 180,E1 -21692.118,E2 -21692.118} C_VEL
LIN {X 0,Y 190.281,Z 466.701,A -85,B 0,C 180,E1 -21694.239,E2 -21694.239} C_VEL
LIN {X 0,Y 190.366,Z 466.479,A -85,B 0,C 180,E1 -21696.362,E2 -21696.362} C_VEL
LIN {X 0,Y 190.689,Z 465.815,A -85,B 0,C 180,E1 -21698.48,E2 -21698.48} C_VEL
LIN {X 0,Y 191.228,Z 464.693,A -85,B 0,C 180,E1 -21700.591,E2 -21700.591} C_VEL
LIN {X 0,Y 192.489,Z 461.939,A -85,B 0,C 180,E1 -21703.731,E2 -21703.731} C_VEL
LIN {X 0,Y 194.329,Z 457.989,A -85,B 0,C 180,E1 -21706.82,E2 -21706.82} C_VEL
LIN {X 0,Y 196.878,Z 452.708,A -85,B 0,C 180,E1 -21709.826,E2 -21709.826} C_VEL
LIN {X 0,Y 199.986,Z 445.82,A -85,B 0,C 180,E1 -21712.744,E2 -21712.744} C_VEL
LIN {X 0,Y 202.034,Z 439.313,A -85,B 0,C 180,E1 -21714.956,E2 -21714.956} C_VEL
LIN {X 0,Y 203.401,Z 431.562,A -85,B 0,C 180,E1 -21717.249,E2 -21717.249} C_VEL
LIN {X 0,Y 203.95,Z 424.117,A -85,B 0,C 180,E1 -21719.231,E2 -21719.231} C_VEL
LIN {X 0,Y 203.77,Z 416.283,A -85,B 0,C 180,E1 -21721.157,E2 -21721.157} C_VEL
LIN {X 0,Y 202.738,Z 406.901,A -85,B 0,C 180,E1 -21723.309,E2 -21723.309} C_VEL
LIN {X 0,Y 200.809,Z 397.339,A -85,B 0,C 180,E1 -21725.463,E2 -21725.463} C_VEL
LIN {X 0,Y 198.997,Z 392.42,A -85,B 0,C 180,E1 -21726.71,E2 -21726.71} C_VEL
LIN {X 0,Y 197.443,Z 388.542,A -85,B 0,C 180,E1 -21727.689,E2 -21727.689} C_VEL
LIN {X 0,Y 195.631,Z 385.42,A -85,B 0,C 180,E1 -21728.706,E2 -21728.706} C_VEL
LIN {X 0,Y 194.991,Z 383.328,A -85,B 0,C 180,E1 -21729.184,E2 -21729.184} C_VEL
LIN {X 0,Y 194.464,Z 380.269,A -85,B 0,C 180,E1 -21733.711,E2 -21733.711} C_VEL
LIN {X 0,Y 194.171,Z 378.558,A -85,B 0,C 180,E1 -21736.549,E2 -21736.549} C_VEL
LIN {X 0,Y 193.903,Z 376.878,A -85,B 0,C 180,E1 -21739.569,E2 -21739.569} C_VEL
LIN {X 0,Y 193.519,Z 374.508,A -85,B 0,C 180,E1 -21744.472,E2 -21744.472} C_VEL
LIN {X 0,Y 193.397,Z 373.458,A -85,B 0,C 180,E1 -21746.967,E2 -21746.967} C_VEL
LIN {X 0,Y 193.094,Z 371.817,A -85,B 0,C 180,E1 -21751.759,E2 -21751.759} C_VEL
LIN {X 0,Y 192.925,Z 370.634,A -85,B 0,C 180,E1 -21756.375,E2 -21756.375} C_VEL
LIN {X 0,Y 192.82,Z 369.798,A -85,B 0,C 180,E1 -21761.388,E2 -21761.388} C_VEL
LIN {X 0,Y 192.804,Z 369.469,A -85,B 0,C 180,E1 -21765.215,E2 -21765.215} C_VEL
LIN {X 0,Y 192.976,Z 369.377,A -85,B 0,C 180,E1 -21769.531,E2 -21769.531} C_VEL
LIN {X 0,Y 193.027,Z 369.635,A -85,B 0,C 180,E1 -21773.727,E2 -21773.727} C_VEL
LIN {X 0,Y 193.421,Z 370.116,A -85,B 0,C 180,E1 -21777.916,E2 -21777.916} C_VEL
LIN {X 0,Y 193.673,Z 370.45,A -85,B 0,C 180,E1 -21779.998,E2 -21779.998} C_VEL
LIN {X 0,Y 193.408,Z 371.495,A -85,B 0,C 180,E1 -21784.166,E2 -21784.166} C_VEL
LIN {X 0,Y 193.583,Z 372.714,A -85,B 0,C 180,E1 -21788.348,E2 -21788.348} C_VEL
LIN {X 0,Y 193.648,Z 373.512,A -85,B 0,C 180,E1 -21790.502,E2 -21790.502} C_VEL
LIN {X 0,Y 194.765,Z 376.354,A -85,B 0,C 180,E1 -21791.277,E2 -21791.277} C_VEL
LIN {X 0,Y 196.509,Z 378.879,A -85,B 0,C 180,E1 -21792.261,E2 -21792.261} C_VEL
LIN {X 0,Y 200.653,Z 387.2,A -85,B 0,C 180,E1 -21794.902,E2 -21794.902} C_VEL
LIN {X 0,Y 203.379,Z 394.666,A -85,B 0,C 180,E1 -21797.079,E2 -21797.079} C_VEL
LIN {X 0,Y 205.492,Z 403.127,A -85,B 0,C 180,E1 -21799.477,E2 -21799.477} C_VEL
LIN {X 0,Y 206.544,Z 411.866,A -85,B 0,C 180,E1 -21801.978,E2 -21801.978} C_VEL
LIN {X 0,Y 206.569,Z 418.716,A -85,B 0,C 180,E1 -21804.094,E2 -21804.094} C_VEL
LIN {X 0,Y 203.797,Z 426.215,A -85,B 0,C 180,E1 -21806.278,E2 -21806.278} C_VEL
LIN {X 0,Y 200.727,Z 433.247,A -85,B 0,C 180,E1 -21808.913,E2 -21808.913} C_VEL
LIN {X 0,Y 198.537,Z 437.747,A -85,B 0,C 180,E1 -21811.051,E2 -21811.051} C_VEL
LIN {X 0,Y 196.584,Z 441.485,A -85,B 0,C 180,E1 -21813.294,E2 -21813.294} C_VEL
LIN {X 0,Y 194.535,Z 445.045,A -85,B 0,C 180,E1 -21816.147,E2 -21816.147} C_VEL
LIN {X 0,Y 193.33,Z 446.875,A -85,B 0,C 180,E1 -21818.166,E2 -21818.166} C_VEL
LIN {X 0,Y 192.449,Z 448.112,A -85,B 0,C 180,E1 -21819.921,E2 -21819.921} C_VEL
LIN {X 0,Y 191.362,Z 449.22,A -85,B 0,C 180,E1 -21822.73,E2 -21822.73} C_VEL
LIN {X 0,Y 190.606,Z 449.447,A -85,B 0,C 180,E1 -21825.524,E2 -21825.524} C_VEL
LIN {X 0,Y 190.201,Z 448.815,A -85,B 0,C 180,E1 -21828.306,E2 -21828.306} C_VEL
LIN {X 0,Y 190.084,Z 447.347,A -85,B 0,C 180,E1 -21831.054,E2 -21831.054} C_VEL
LIN {X 0,Y 190.367,Z 444.431,A -85,B 0,C 180,E1 -21834.307,E2 -21834.307} C_VEL
LIN {X 0,Y 191.043,Z 439.865,A -85,B 0,C 180,E1 -21837.786,E2 -21837.786} C_VEL
LIN {X 0,Y 191.996,Z 434.227,A -85,B 0,C 180,E1 -21840.91,E2 -21840.91} C_VEL
LIN {X 0,Y 193.103,Z 428.015,A -85,B 0,C 180,E1 -21843.52,E2 -21843.52} C_VEL
LIN {X 0,Y 194.075,Z 422.256,A -85,B 0,C 180,E1 -21845.506,E2 -21845.506} C_VEL
LIN {X 0,Y 195.293,Z 415.389,A -85,B 0,C 180,E1 -21847.454,E2 -21847.454} C_VEL
LIN {X 0,Y 196.554,Z 407.329,A -85,B 0,C 180,E1 -21849.321,E2 -21849.321} C_VEL
LIN {X 0,Y 197.047,Z 403.085,A -85,B 0,C 180,E1 -21850.192,E2 -21850.192} C_VEL
LIN {X 0,Y 195.766,Z 393.415,A -85,B 0,C 180,E1 -21851.96,E2 -21851.96} C_VEL
LIN {X 0,Y 194.149,Z 383.526,A -85,B 0,C 180,E1 -21853.435,E2 -21853.435} C_VEL
LIN {X 0,Y 192.217,Z 373.537,A -85,B 0,C 180,E1 -21854.626,E2 -21854.626} C_VEL
LIN {X 0,Y 191.511,Z 369.93,A -85,B 0,C 180,E1 -21855.044,E2 -21855.044} C_VEL
LIN {X 0,Y 191.672,Z 369.429,A -85,B 0,C 180,E1 -21856.209,E2 -21856.209} C_VEL
LIN {X 0,Y 192.649,Z 369.301,A -85,B 0,C 180,E1 -21861.607,E2 -21861.607} C_VEL
LIN {X 0,Y 192.926,Z 369.268,A -85,B 0,C 180,E1 -21865.819,E2 -21865.819} C_VEL
LIN {X 0,Y 193.434,Z 369.205,A -85,B 0,C 180,E1 -21869.997,E2 -21869.997} C_VEL
LIN {X 0,Y 192.973,Z 369.261,A -85,B 0,C 180,E1 -21874.174,E2 -21874.174} C_VEL
LIN {X 0,Y 193.07,Z 369.247,A -85,B 0,C 180,E1 -21878.37,E2 -21878.37} C_VEL
LIN {X 0,Y 192.844,Z 369.272,A -85,B 0,C 180,E1 -21882.628,E2 -21882.628} C_VEL
LIN {X 0,Y 192.747,Z 369.287,A -85,B 0,C 180,E1 -21886.957,E2 -21886.957} C_VEL
LIN {X 0,Y 192.626,Z 369.301,A -85,B 0,C 180,E1 -21891.395,E2 -21891.395} C_VEL
LIN {X 0,Y 192.653,Z 369.299,A -85,B 0,C 180,E1 -21894.223,E2 -21894.223} C_VEL
LIN {X 0,Y 192.638,Z 369.297,A -85,B 0,C 180,E1 -21898.891,E2 -21898.891} C_VEL
LIN {X 0,Y 192.588,Z 369.309,A -85,B 0,C 180,E1 -21903.184,E2 -21903.184} C_VEL
LIN {X 0,Y 192.616,Z 369.301,A -85,B 0,C 180,E1 -21908.333,E2 -21908.333} C_VEL
LIN {X 0,Y 192.622,Z 369.302,A -85,B 0,C 180,E1 -21913.141,E2 -21913.141} C_VEL
LIN {X 0,Y 192.621,Z 369.303,A -85,B 0,C 180,E1 -21916.859,E2 -21916.859} C_VEL
LIN {X 0,Y 192.6,Z 369.303,A -85,B 0,C 180,E1 -21921.663,E2 -21921.663} C_VEL
LIN {X 0,Y 192.588,Z 369.309,A -85,B 0,C 180,E1 -21926.815,E2 -21926.815} C_VEL
LIN {X 0,Y 192.653,Z 369.295,A -85,B 0,C 180,E1 -21931.693,E2 -21931.693} C_VEL
LIN {X 0,Y 192.705,Z 369.294,A -85,B 0,C 180,E1 -21936.351,E2 -21936.351} C_VEL
LIN {X 0,Y 192.771,Z 369.282,A -85,B 0,C 180,E1 -21941.414,E2 -21941.414} C_VEL
LIN {X 0,Y 192.843,Z 369.271,A -85,B 0,C 180,E1 -21947.372,E2 -21947.372} C_VEL
LIN {X 0,Y 193.068,Z 369.247,A -85,B 0,C 180,E1 -21951.63,E2 -21951.63} C_VEL
LIN {X 0,Y 193.255,Z 369.224,A -85,B 0,C 180,E1 -21957.918,E2 -21957.918} C_VEL
LIN {X 0,Y 193.434,Z 369.204,A -85,B 0,C 180,E1 -21960.002,E2 -21960.002} C_VEL
LIN {X 0,Y 192.972,Z 369.257,A -85,B 0,C 180,E1 -21964.179,E2 -21964.179} C_VEL
LIN {X 0,Y 193.07,Z 369.247,A -85,B 0,C 180,E1 -21968.374,E2 -21968.374} C_VEL
LIN {X 0,Y 193.002,Z 369.254,A -85,B 0,C 180,E1 -21970.541,E2 -21970.541} C_VEL
LIN {X 0,Y 192.763,Z 369.285,A -85,B 0,C 180,E1 -21976.96,E2 -21976.96} C_VEL
LIN {X 0,Y 192.636,Z 369.299,A -85,B 0,C 180,E1 -21981.399,E2 -21981.399} C_VEL
LIN {X 0,Y 192.658,Z 369.298,A -85,B 0,C 180,E1 -21984.227,E2 -21984.227} C_VEL
LIN {X 0,Y 192.644,Z 369.298,A -85,B 0,C 180,E1 -21988.895,E2 -21988.895} C_VEL
LIN {X 0,Y 192.594,Z 369.309,A -85,B 0,C 180,E1 -21993.189,E2 -21993.189} C_VEL
LIN {X 0,Y 192.547,Z 369.309,A -85,B 0,C 180,E1 -21998.355,E2 -21998.355} C_VEL
LIN {X 0,Y 192.534,Z 369.312,A -85,B 0,C 180,E1 -22003.914,E2 -22003.914} C_VEL
LIN {X 0,Y 192.75,Z 369.46,A -85,B 0,C 180,E1 -22006.493,E2 -22006.493} C_VEL
LIN {X 0,Y 193.646,Z 374.13,A -85,B 0,C 180,E1 -22011.908,E2 -22011.908} C_VEL
LIN {X 0,Y 194.044,Z 376.541,A -85,B 0,C 180,E1 -22014.589,E2 -22014.589} C_VEL
LIN {X 0,Y 193.782,Z 378.855,A -85,B 0,C 180,E1 -22017.046,E2 -22017.046} C_VEL
LIN {X 0,Y 192.511,Z 383.366,A -85,B 0,C 180,E1 -22021.671,E2 -22021.671} C_VEL
LIN {X 0,Y 191.811,Z 386.687,A -85,B 0,C 180,E1 -22025.011,E2 -22025.011} C_VEL
LIN {X 0,Y 193.192,Z 399.326,A -85,B 0,C 180,E1 -22026.26,E2 -22026.26} C_VEL
LIN {X 0,Y 193.833,Z 407.635,A -85,B 0,C 180,E1 -22027.344,E2 -22027.344} C_VEL
LIN {X 0,Y 194.371,Z 416.657,A -85,B 0,C 180,E1 -22028.806,E2 -22028.806} C_VEL
LIN {X 0,Y 194.586,Z 425.041,A -85,B 0,C 180,E1 -22030.457,E2 -22030.457} C_VEL
LIN {X 0,Y 194.538,Z 432.118,A -85,B 0,C 180,E1 -22032.12,E2 -22032.12} C_VEL
LIN {X 0,Y 193.546,Z 437.813,A -85,B 0,C 180,E1 -22033.658,E2 -22033.658} C_VEL
LIN {X 0,Y 192.489,Z 444.193,A -85,B 0,C 180,E1 -22035.735,E2 -22035.735} C_VEL
LIN {X 0,Y 191.663,Z 449.502,A -85,B 0,C 180,E1 -22037.831,E2 -22037.831} C_VEL
LIN {X 0,Y 190.963,Z 454.883,A -85,B 0,C 180,E1 -22040.47,E2 -22040.47} C_VEL
LIN {X 0,Y 190.613,Z 458.36,A -85,B 0,C 180,E1 -22042.588,E2 -22042.588} C_VEL
LIN {X 0,Y 190.408,Z 462.329,A -85,B 0,C 180,E1 -22045.769,E2 -22045.769} C_VEL
LIN {X 0,Y 190.478,Z 464.231,A -85,B 0,C 180,E1 -22047.888,E2 -22047.888} C_VEL
LIN {X 0,Y 190.478,Z 465.826,A -85,B 0,C 180,E1 -22050.553,E2 -22050.553} C_VEL
LIN {X 0,Y 189.663,Z 466.451,A -85,B 0,C 180,E1 -22052.309,E2 -22052.309} C_VEL
LIN {X 0,Y 186.756,Z 466.561,A -85,B 0,C 180,E1 -22055.198,E2 -22055.198} C_VEL
LIN {X 0,Y 184.186,Z 465.89,A -85,B 0,C 180,E1 -22058.169,E2 -22058.169} C_VEL
LIN {X 0,Y 183.928,Z 465.039,A -85,B 0,C 180,E1 -22060.002,E2 -22060.002} C_VEL
LIN {X 0,Y 185.063,Z 462.91,A -85,B 0,C 180,E1 -22063.174,E2 -22063.174} C_VEL
LIN {X 0,Y 186.847,Z 459.588,A -85,B 0,C 180,E1 -22066.388,E2 -22066.388} C_VEL
LIN {X 0,Y 189.258,Z 454.891,A -85,B 0,C 180,E1 -22069.527,E2 -22069.527} C_VEL
LIN {X 0,Y 191.798,Z 449.829,A -85,B 0,C 180,E1 -22072.063,E2 -22072.063} C_VEL
LIN {X 0,Y 194.044,Z 444.97,A -85,B 0,C 180,E1 -22074.048,E2 -22074.048} C_VEL
LIN {X 0,Y 195.946,Z 438.702,A -85,B 0,C 180,E1 -22076.273,E2 -22076.273} C_VEL
LIN {X 0,Y 197.112,Z 432.615,A -85,B 0,C 180,E1 -22078.195,E2 -22078.195} C_VEL
LIN {X 0,Y 197.811,Z 425.437,A -85,B 0,C 180,E1 -22080.231,E2 -22080.231} C_VEL
LIN {X 0,Y 197.74,Z 416.926,A -85,B 0,C 180,E1 -22082.466,E2 -22082.466} C_VEL
LIN {X 0,Y 197.037,Z 408.915,A -85,B 0,C 180,E1 -22084.466,E2 -22084.466} C_VEL
LIN {X 0,Y 195.583,Z 400.829,A -85,B 0,C 180,E1 -22086.453,E2 -22086.453} C_VEL
LIN {X 0,Y 193.099,Z 393.51,A -85,B 0,C 180,E1 -22088.505,E2 -22088.505} C_VEL
LIN {X 0,Y 191.25,Z 389.971,A -85,B 0,C 180,E1 -22089.664,E2 -22089.664} C_VEL
LIN {X 0,Y 190.508,Z 388.333,A -85,B 0,C 180,E1 -22090.175,E2 -22090.175} C_VEL
LIN {X 0,Y 188.294,Z 384.847,A -85,B 0,C 180,E1 -22091.535,E2 -22091.535} C_VEL
LIN {X 0,Y 187.643,Z 382.741,A -85,B 0,C 180,E1 -22092.071,E2 -22092.071} C_VEL
LIN {X 0,Y 187.297,Z 380.676,A -85,B 0,C 180,E1 -22095.478,E2 -22095.478} C_VEL
LIN {X 0,Y 186.889,Z 378.101,A -85,B 0,C 180,E1 -22100.259,E2 -22100.259} C_VEL
LIN {X 0,Y 186.732,Z 376.8,A -85,B 0,C 180,E1 -22102.971,E2 -22102.971} C_VEL
LIN {X 0,Y 186.367,Z 374.727,A -85,B 0,C 180,E1 -22108.131,E2 -22108.131} C_VEL
LIN {X 0,Y 186.266,Z 373.879,A -85,B 0,C 180,E1 -22110.624,E2 -22110.624} C_VEL
LIN {X 0,Y 186.069,Z 372.58,A -85,B 0,C 180,E1 -22115.448,E2 -22115.448} C_VEL
LIN {X 0,Y 185.936,Z 371.621,A -85,B 0,C 180,E1 -22120.907,E2 -22120.907} C_VEL
LIN {X 0,Y 185.921,Z 371.255,A -85,B 0,C 180,E1 -22124.654,E2 -22124.654} C_VEL
LIN {X 0,Y 186.062,Z 371.113,A -85,B 0,C 180,E1 -22129.15,E2 -22129.15} C_VEL
LIN {X 0,Y 186.156,Z 371.168,A -85,B 0,C 180,E1 -22131.312,E2 -22131.312} C_VEL
LIN {X 0,Y 186.515,Z 371.775,A -85,B 0,C 180,E1 -22137.838,E2 -22137.838} C_VEL
LIN {X 0,Y 186.764,Z 372.089,A -85,B 0,C 180,E1 -22139.998,E2 -22139.998} C_VEL
LIN {X 0,Y 186.482,Z 373.137,A -85,B 0,C 180,E1 -22144.321,E2 -22144.321} C_VEL
LIN {X 0,Y 186.631,Z 374.172,A -85,B 0,C 180,E1 -22147.639,E2 -22147.639} C_VEL
LIN {X 0,Y 187.772,Z 376.888,A -85,B 0,C 180,E1 -22148.54,E2 -22148.54} C_VEL
LIN {X 0,Y 189.768,Z 379.418,A -85,B 0,C 180,E1 -22149.793,E2 -22149.793} C_VEL
LIN {X 0,Y 191.512,Z 382.757,A -85,B 0,C 180,E1 -22150.97,E2 -22150.97} C_VEL
LIN {X 0,Y 195.463,Z 390.86,A -85,B 0,C 180,E1 -22153.87,E2 -22153.87} C_VEL
LIN {X 0,Y 198.201,Z 399.054,A -85,B 0,C 180,E1 -22156.477,E2 -22156.477} C_VEL
LIN {X 0,Y 199.826,Z 407.109,A -85,B 0,C 180,E1 -22158.983,E2 -22158.983} C_VEL
LIN {X 0,Y 200.423,Z 415.389,A -85,B 0,C 180,E1 -22161.602,E2 -22161.602} C_VEL
LIN {X 0,Y 200.37,Z 419.791,A -85,B 0,C 180,E1 -22163.048,E2 -22163.048} C_VEL
LIN {X 0,Y 199.117,Z 423.535,A -85,B 0,C 180,E1 -22164.196,E2 -22164.196} C_VEL
LIN {X 0,Y 195.698,Z 431.391,A -85,B 0,C 180,E1 -22166.885,E2 -22166.885} C_VEL
LIN {X 0,Y 193.156,Z 436.474,A -85,B 0,C 180,E1 -22169.158,E2 -22169.158} C_VEL
LIN {X 0,Y 190.493,Z 441.252,A -85,B 0,C 180,E1 -22171.941,E2 -22171.941} C_VEL
LIN {X 0,Y 188.258,Z 444.868,A -85,B 0,C 180,E1 -22174.781,E2 -22174.781} C_VEL
LIN {X 0,Y 186.443,Z 447.43,A -85,B 0,C 180,E1 -22177.661,E2 -22177.661} C_VEL
LIN {X 0,Y 185.064,Z 449.031,A -85,B 0,C 180,E1 -22180.575,E2 -22180.575} C_VEL
LIN {X 0,Y 184.029,Z 449.724,A -85,B 0,C 180,E1 -22183.477,E2 -22183.477} C_VEL
LIN {X 0,Y 183.27,Z 449.479,A -85,B 0,C 180,E1 -22186.766,E2 -22186.766} C_VEL
LIN {X 0,Y 182.976,Z 448.084,A -85,B 0,C 180,E1 -22190.187,E2 -22190.187} C_VEL
LIN {X 0,Y 183.174,Z 445.298,A -85,B 0,C 180,E1 -22193.676,E2 -22193.676} C_VEL
LIN {X 0,Y 183.591,Z 442.483,A -85,B 0,C 180,E1 -22196.169,E2 -22196.169} C_VEL
LIN {X 0,Y 184.261,Z 438.237,A -85,B 0,C 180,E1 -22199.006,E2 -22199.006} C_VEL
LIN {X 0,Y 185.073,Z 433.577,A -85,B 0,C 180,E1 -22201.472,E2 -22201.472} C_VEL
LIN {X 0,Y 186.129,Z 427.814,A -85,B 0,C 180,E1 -22203.93,E2 -22203.93} C_VEL
LIN {X 0,Y 187.28,Z 421.246,A -85,B 0,C 180,E1 -22206.206,E2 -22206.206} C_VEL
LIN {X 0,Y 188.492,Z 414.562,A -85,B 0,C 180,E1 -22208.106,E2 -22208.106} C_VEL
LIN {X 0,Y 189.788,Z 406.593,A -85,B 0,C 180,E1 -22209.966,E2 -22209.966} C_VEL
LIN {X 0,Y 190.074,Z 403.828,A -85,B 0,C 180,E1 -22210.56,E2 -22210.56} C_VEL
LIN {X 0,Y 188.829,Z 394.303,A -85,B 0,C 180,E1 -22212.395,E2 -22212.395} C_VEL
LIN {X 0,Y 187.593,Z 386.337,A -85,B 0,C 180,E1 -22213.679,E2 -22213.679} C_VEL
LIN {X 0,Y 185.629,Z 375.787,A -85,B 0,C 180,E1 -22215.05,E2 -22215.05} C_VEL
LIN {X 0,Y 184.51,Z 370.321,A -85,B 0,C 180,E1 -22215.663,E2 -22215.663} C_VEL
LIN {X 0,Y 185.53,Z 370.187,A -85,B 0,C 180,E1 -22221.282,E2 -22221.282} C_VEL
LIN {X 0,Y 185.78,Z 370.157,A -85,B 0,C 180,E1 -22223.481,E2 -22223.481} C_VEL
LIN {X 0,Y 186.188,Z 370.107,A -85,B 0,C 180,E1 -22227.834,E2 -22227.834} C_VEL
LIN {X 0,Y 186.398,Z 370.081,A -85,B 0,C 180,E1 -22229.997,E2 -22229.997} C_VEL
LIN {X 0,Y 185.921,Z 370.139,A -85,B 0,C 180,E1 -22234.333,E2 -22234.333} C_VEL
LIN {X 0,Y 186.02,Z 370.124,A -85,B 0,C 180,E1 -22238.689,E2 -22238.689} C_VEL
LIN {X 0,Y 185.755,Z 370.155,A -85,B 0,C 180,E1 -22243.118,E2 -22243.118} C_VEL
LIN {X 0,Y 185.68,Z 370.169,A -85,B 0,C 180,E1 -22247.623,E2 -22247.623} C_VEL
LIN {X 0,Y 185.586,Z 370.178,A -85,B 0,C 180,E1 -22252.249,E2 -22252.249} C_VEL
LIN {X 0,Y 185.551,Z 370.182,A -85,B 0,C 180,E1 -22257.03,E2 -22257.03} C_VEL
LIN {X 0,Y 185.567,Z 370.181,A -85,B 0,C 180,E1 -22259.492,E2 -22259.492} C_VEL
LIN {X 0,Y 185.51,Z 370.187,A -85,B 0,C 180,E1 -22264.626,E2 -22264.626} C_VEL
LIN {X 0,Y 185.556,Z 370.181,A -85,B 0,C 180,E1 -22267.313,E2 -22267.313} C_VEL
LIN {X 0,Y 185.583,Z 370.18,A -85,B 0,C 180,E1 -22270.769,E2 -22270.769} C_VEL
LIN {X 0,Y 185.575,Z 370.178,A -85,B 0,C 180,E1 -22276.013,E2 -22276.013} C_VEL
LIN {X 0,Y 185.554,Z 370.182,A -85,B 0,C 180,E1 -22279.921,E2 -22279.921} C_VEL
LIN {X 0,Y 185.563,Z 370.18,A -85,B 0,C 180,E1 -22282.704,E2 -22282.704} C_VEL
LIN {X 0,Y 185.533,Z 370.185,A -85,B 0,C 180,E1 -22287.976,E2 -22287.976} C_VEL
LIN {X 0,Y 185.57,Z 370.179,A -85,B 0,C 180,E1 -22290.576,E2 -22290.576} C_VEL
LIN {X 0,Y 185.612,Z 370.176,A -85,B 0,C 180,E1 -22295.389,E2 -22295.389} C_VEL
LIN {X 0,Y 185.7,Z 370.163,A -85,B 0,C 180,E1 -22301.101,E2 -22301.101} C_VEL
LIN {X 0,Y 185.722,Z 370.163,A -85,B 0,C 180,E1 -22304.642,E2 -22304.642} C_VEL
LIN {X 0,Y 185.932,Z 370.134,A -85,B 0,C 180,E1 -22309.33,E2 -22309.33} C_VEL
LIN {X 0,Y 185.959,Z 370.132,A -85,B 0,C 180,E1 -22313.492,E2 -22313.492} C_VEL
LIN {X 0,Y 186.199,Z 370.102,A -85,B 0,C 180,E1 -22317.839,E2 -22317.839} C_VEL
LIN {X 0,Y 186.397,Z 370.081,A -85,B 0,C 180,E1 -22320.002,E2 -22320.002} C_VEL
LIN {X 0,Y 185.92,Z 370.134,A -85,B 0,C 180,E1 -22324.338,E2 -22324.338} C_VEL
LIN {X 0,Y 186.021,Z 370.125,A -85,B 0,C 180,E1 -22328.694,E2 -22328.694} C_VEL
LIN {X 0,Y 185.735,Z 370.156,A -85,B 0,C 180,E1 -22333.125,E2 -22333.125} C_VEL
LIN {X 0,Y 185.687,Z 370.166,A -85,B 0,C 180,E1 -22338.887,E2 -22338.887} C_VEL
LIN {X 0,Y 185.595,Z 370.178,A -85,B 0,C 180,E1 -22344.665,E2 -22344.665} C_VEL
LIN {X 0,Y 185.574,Z 370.179,A -85,B 0,C 180,E1 -22349.496,E2 -22349.496} C_VEL
LIN {X 0,Y 185.494,Z 370.191,A -85,B 0,C 180,E1 -22354.635,E2 -22354.635} C_VEL
LIN {X 0,Y 185.501,Z 370.187,A -85,B 0,C 180,E1 -22357.316,E2 -22357.316} C_VEL
LIN {X 0,Y 185.468,Z 370.195,A -85,B 0,C 180,E1 -22360.728,E2 -22360.728} C_VEL
LIN {X 0,Y 185.695,Z 370.224,A -85,B 0,C 180,E1 -22366.267,E2 -22366.267} C_VEL
LIN {X 0,Y 186.667,Z 375.188,A -85,B 0,C 180,E1 -22372.249,E2 -22372.249} C_VEL
LIN {X 0,Y 186.952,Z 377.026,A -85,B 0,C 180,E1 -22374.364,E2 -22374.364} C_VEL
LIN {X 0,Y 186.695,Z 379.422,A -85,B 0,C 180,E1 -22377.009,E2 -22377.009} C_VEL
LIN {X 0,Y 185.1,Z 384.954,A -85,B 0,C 180,E1 -22382.898,E2 -22382.898} C_VEL
LIN {X 0,Y 184.824,Z 386.478,A -85,B 0,C 180,E1 -22384.364,E2 -22384.364} C_VEL
LIN {X 0,Y 186.208,Z 398.947,A -85,B 0,C 180,E1 -22385.657,E2 -22385.657} C_VEL
LIN {X 0,Y 186.928,Z 409.08,A -85,B 0,C 180,E1 -22387.074,E2 -22387.074} C_VEL
LIN {X 0,Y 187.372,Z 417.266,A -85,B 0,C 180,E1 -22388.491,E2 -22388.491} C_VEL
LIN {X 0,Y 187.528,Z 423.993,A -85,B 0,C 180,E1 -22389.864,E2 -22389.864} C_VEL
LIN {X 0,Y 187.547,Z 431.619,A -85,B 0,C 180,E1 -22391.712,E2 -22391.712} C_VEL
LIN {X 0,Y 186.428,Z 438.197,A -85,B 0,C 180,E1 -22393.579,E2 -22393.579} C_VEL
LIN {X 0,Y 185.364,Z 444.459,A -85,B 0,C 180,E1 -22395.736,E2 -22395.736} C_VEL
LIN {X 0,Y 184.508,Z 449.659,A -85,B 0,C 180,E1 -22397.91,E2 -22397.91} C_VEL
LIN {X 0,Y 183.946,Z 453.996,A -85,B 0,C 180,E1 -22400.103,E2 -22400.103} C_VEL
LIN {X 0,Y 183.462,Z 459.097,A -85,B 0,C 180,E1 -22403.404,E2 -22403.404} C_VEL
LIN {X 0,Y 183.314,Z 462.568,A -85,B 0,C 180,E1 -22406.488,E2 -22406.488} C_VEL
LIN {X 0,Y 183.479,Z 465.132,A -85,B 0,C 180,E1 -22410.003,E2 -22410.003} C_VEL
LIN {X 0,Y 183.301,Z 466,A -85,B 0,C 180,E1 -22412.2,E2 -22412.2} C_VEL
LIN {X 0,Y 183.193,Z 466.314,A -85,B 0,C 180,E1 -22414.403,E2 -22414.403} C_VEL
LIN {X 0,Y 183.308,Z 466.185,A -85,B 0,C 180,E1 -22416.608,E2 -22416.608} C_VEL
LIN {X 0,Y 183.928,Z 465.039,A -85,B 0,C 180,E1 -22420.002,E2 -22420.002} C_VEL
LIN {X 0,Y 183.838,Z 464.035,A -85,B 0,C 180,E1 -22421.816,E2 -22421.816} C_VEL
LIN {X 0,Y 182.271,Z 461.715,A -85,B 0,C 180,E1 -22424.799,E2 -22424.799} C_VEL
LIN {X 0,Y 181.201,Z 458.681,A -85,B 0,C 180,E1 -22427.751,E2 -22427.751} C_VEL
LIN {X 0,Y 181.876,Z 456.358,A -85,B 0,C 180,E1 -22429.458,E2 -22429.458} C_VEL
LIN {X 0,Y 185.255,Z 450.287,A -85,B 0,C 180,E1 -22432.886,E2 -22432.886} C_VEL
LIN {X 0,Y 188.104,Z 444.219,A -85,B 0,C 180,E1 -22435.449,E2 -22435.449} C_VEL
LIN {X 0,Y 189.885,Z 438.357,A -85,B 0,C 180,E1 -22437.609,E2 -22437.609} C_VEL
LIN {X 0,Y 191.137,Z 431.771,A -85,B 0,C 180,E1 -22439.764,E2 -22439.764} C_VEL
LIN {X 0,Y 191.781,Z 423.819,A -85,B 0,C 180,E1 -22442.146,E2 -22442.146} C_VEL
LIN {X 0,Y 191.752,Z 416.13,A -85,B 0,C 180,E1 -22444.279,E2 -22444.279} C_VEL
LIN {X 0,Y 191.206,Z 409.611,A -85,B 0,C 180,E1 -22446.035,E2 -22446.035} C_VEL
LIN {X 0,Y 189.93,Z 402.516,A -85,B 0,C 180,E1 -22448.003,E2 -22448.003} C_VEL
LIN {X 0,Y 188.426,Z 398.146,A -85,B 0,C 180,E1 -22449.354,E2 -22449.354} C_VEL
LIN {X 0,Y 186.338,Z 393.471,A -85,B 0,C 180,E1 -22451.031,E2 -22451.031} C_VEL
LIN {X 0,Y 184.182,Z 389.496,A -85,B 0,C 180,E1 -22452.586,E2 -22452.586} C_VEL
LIN {X 0,Y 183.593,Z 388.095,A -85,B 0,C 180,E1 -22453.079,E2 -22453.079} C_VEL
LIN {X 0,Y 181.244,Z 384.706,A -85,B 0,C 180,E1 -22454.758,E2 -22454.758} C_VEL
LIN {X 0,Y 180.341,Z 382.067,A -85,B 0,C 180,E1 -22455.625,E2 -22455.625} C_VEL
LIN {X 0,Y 180.098,Z 380.571,A -85,B 0,C 180,E1 -22458.438,E2 -22458.438} C_VEL
LIN {X 0,Y 179.875,Z 379.127,A -85,B 0,C 180,E1 -22461.396,E2 -22461.396} C_VEL
LIN {X 0,Y 179.65,Z 377.491,A -85,B 0,C 180,E1 -22465.243,E2 -22465.243} C_VEL
LIN {X 0,Y 179.397,Z 375.946,A -85,B 0,C 180,E1 -22469.531,E2 -22469.531} C_VEL
LIN {X 0,Y 179.189,Z 374.577,A -85,B 0,C 180,E1 -22474.439,E2 -22474.439} C_VEL
LIN {X 0,Y 179.024,Z 373.633,A -85,B 0,C 180,E1 -22479.308,E2 -22479.308} C_VEL
LIN {X 0,Y 179.028,Z 373.072,A -85,B 0,C 180,E1 -22484.048,E2 -22484.048} C_VEL
LIN {X 0,Y 179.133,Z 372.875,A -85,B 0,C 180,E1 -22488.777,E2 -22488.777} C_VEL
LIN {X 0,Y 179.25,Z 372.883,A -85,B 0,C 180,E1 -22490.975,E2 -22490.975} C_VEL
LIN {X 0,Y 179.594,Z 373.434,A -85,B 0,C 180,E1 -22497.755,E2 -22497.755} C_VEL
LIN {X 0,Y 179.862,Z 373.744,A -85,B 0,C 180,E1 -22499.998,E2 -22499.998} C_VEL
LIN {X 0,Y 179.577,Z 374.708,A -85,B 0,C 180,E1 -22504.136,E2 -22504.136} C_VEL
LIN {X 0,Y 180.617,Z 377.391,A -85,B 0,C 180,E1 -22505.16,E2 -22505.16} C_VEL
LIN {X 0,Y 183.11,Z 380.34,A -85,B 0,C 180,E1 -22506.956,E2 -22506.956} C_VEL
LIN {X 0,Y 184.591,Z 383.168,A -85,B 0,C 180,E1 -22508.131,E2 -22508.131} C_VEL
LIN {X 0,Y 186.045,Z 385.44,A -85,B 0,C 180,E1 -22509.236,E2 -22509.236} C_VEL
LIN {X 0,Y 189.699,Z 393.097,A -85,B 0,C 180,E1 -22512.298,E2 -22512.298} C_VEL
LIN {X 0,Y 192.072,Z 400.208,A -85,B 0,C 180,E1 -22514.838,E2 -22514.838} C_VEL
LIN {X 0,Y 193.689,Z 407.803,A -85,B 0,C 180,E1 -22517.416,E2 -22517.416} C_VEL
LIN {X 0,Y 194.279,Z 414.971,A -85,B 0,C 180,E1 -22519.851,E2 -22519.851} C_VEL
LIN {X 0,Y 194.038,Z 421.961,A -85,B 0,C 180,E1 -22522.35,E2 -22522.35} C_VEL
LIN {X 0,Y 191.192,Z 428.59,A -85,B 0,C 180,E1 -22524.521,E2 -22524.521} C_VEL
LIN {X 0,Y 188.642,Z 433.753,A -85,B 0,C 180,E1 -22526.597,E2 -22526.597} C_VEL
LIN {X 0,Y 186.29,Z 438.016,A -85,B 0,C 180,E1 -22528.697,E2 -22528.697} C_VEL
LIN {X 0,Y 184.139,Z 441.616,A -85,B 0,C 180,E1 -22530.898,E2 -22530.898} C_VEL
LIN {X 0,Y 181.681,Z 445.308,A -85,B 0,C 180,E1 -22533.921,E2 -22533.921} C_VEL
LIN {X 0,Y 180.408,Z 447.054,A -85,B 0,C 180,E1 -22535.753,E2 -22535.753} C_VEL
LIN {X 0,Y 178.591,Z 449.069,A -85,B 0,C 180,E1 -22539.02,E2 -22539.02} C_VEL
LIN {X 0,Y 177.235,Z 450.029,A -85,B 0,C 180,E1 -22542.381,E2 -22542.381} C_VEL
LIN {X 0,Y 176.693,Z 450.173,A -85,B 0,C 180,E1 -22544.275,E2 -22544.275} C_VEL
LIN {X 0,Y 176.092,Z 449.596,A -85,B 0,C 180,E1 -22547.271,E2 -22547.271} C_VEL
LIN {X 0,Y 175.893,Z 448.174,A -85,B 0,C 180,E1 -22550.257,E2 -22550.257} C_VEL
LIN {X 0,Y 176.011,Z 445.91,A -85,B 0,C 180,E1 -22553.203,E2 -22553.203} C_VEL
LIN {X 0,Y 176.583,Z 441.967,A -85,B 0,C 180,E1 -22556.694,E2 -22556.694} C_VEL
LIN {X 0,Y 177.385,Z 437.209,A -85,B 0,C 180,E1 -22559.819,E2 -22559.819} C_VEL
LIN {X 0,Y 178.298,Z 432.194,A -85,B 0,C 180,E1 -22562.407,E2 -22562.407} C_VEL
LIN {X 0,Y 179.565,Z 425.668,A -85,B 0,C 180,E1 -22565.116,E2 -22565.116} C_VEL
LIN {X 0,Y 181.017,Z 417.432,A -85,B 0,C 180,E1 -22567.812,E2 -22567.812} C_VEL
LIN {X 0,Y 182.547,Z 408.751,A -85,B 0,C 180,E1 -22570.018,E2 -22570.018} C_VEL
LIN {X 0,Y 183.088,Z 404.572,A -85,B 0,C 180,E1 -22570.954,E2 -22570.954} C_VEL
LIN {X 0,Y 181.91,Z 395.12,A -85,B 0,C 180,E1 -22572.864,E2 -22572.864} C_VEL
LIN {X 0,Y 180.37,Z 385.432,A -85,B 0,C 180,E1 -22574.459,E2 -22574.459} C_VEL
LIN {X 0,Y 178.527,Z 375.698,A -85,B 0,C 180,E1 -22575.754,E2 -22575.754} C_VEL
LIN {X 0,Y 177.584,Z 371.182,A -85,B 0,C 180,E1 -22576.334,E2 -22576.334} C_VEL
LIN {X 0,Y 178.41,Z 371.075,A -85,B 0,C 180,E1 -22580.931,E2 -22580.931} C_VEL
LIN {X 0,Y 178.711,Z 371.038,A -85,B 0,C 180,E1 -22583.222,E2 -22583.222} C_VEL
LIN {X 0,Y 179.131,Z 370.986,A -85,B 0,C 180,E1 -22587.749,E2 -22587.749} C_VEL
LIN {X 0,Y 179.361,Z 370.958,A -85,B 0,C 180,E1 -22589.997,E2 -22589.997} C_VEL
LIN {X 0,Y 178.869,Z 371.016,A -85,B 0,C 180,E1 -22594.504,E2 -22594.504} C_VEL
LIN {X 0,Y 178.969,Z 371.003,A -85,B 0,C 180,E1 -22599.034,E2 -22599.034} C_VEL
LIN {X 0,Y 178.677,Z 371.039,A -85,B 0,C 180,E1 -22603.648,E2 -22603.648} C_VEL
LIN {X 0,Y 178.639,Z 371.042,A -85,B 0,C 180,E1 -22608.342,E2 -22608.342} C_VEL
LIN {X 0,Y 178.5,Z 371.062,A -85,B 0,C 180,E1 -22613.183,E2 -22613.183} C_VEL
LIN {X 0,Y 178.475,Z 371.06,A -85,B 0,C 180,E1 -22618.195,E2 -22618.195} C_VEL
LIN {X 0,Y 178.467,Z 371.065,A -85,B 0,C 180,E1 -22620.789,E2 -22620.789} C_VEL
LIN {X 0,Y 178.474,Z 371.064,A -85,B 0,C 180,E1 -22624.219,E2 -22624.219} C_VEL
LIN {X 0,Y 178.483,Z 371.064,A -85,B 0,C 180,E1 -22629.047,E2 -22629.047} C_VEL
LIN {X 0,Y 178.508,Z 371.06,A -85,B 0,C 180,E1 -22632.009,E2 -22632.009} C_VEL
LIN {X 0,Y 178.518,Z 371.057,A -85,B 0,C 180,E1 -22635.119,E2 -22635.119} C_VEL
LIN {X 0,Y 178.506,Z 371.061,A -85,B 0,C 180,E1 -22638.417,E2 -22638.417} C_VEL
LIN {X 0,Y 178.455,Z 371.064,A -85,B 0,C 180,E1 -22643.794,E2 -22643.794} C_VEL
LIN {X 0,Y 178.479,Z 371.066,A -85,B 0,C 180,E1 -22646.548,E2 -22646.548} C_VEL
LIN {X 0,Y 178.511,Z 371.059,A -85,B 0,C 180,E1 -22650.007,E2 -22650.007} C_VEL
LIN {X 0,Y 178.533,Z 371.059,A -85,B 0,C 180,E1 -22654.869,E2 -22654.869} C_VEL
LIN {X 0,Y 178.644,Z 371.043,A -85,B 0,C 180,E1 -22660.755,E2 -22660.755} C_VEL
LIN {X 0,Y 178.668,Z 371.042,A -85,B 0,C 180,E1 -22664.02,E2 -22664.02} C_VEL
LIN {X 0,Y 178.884,Z 371.011,A -85,B 0,C 180,E1 -22669.155,E2 -22669.155} C_VEL
LIN {X 0,Y 178.924,Z 371.008,A -85,B 0,C 180,E1 -22673.235,E2 -22673.235} C_VEL
LIN {X 0,Y 179.145,Z 370.98,A -85,B 0,C 180,E1 -22677.754,E2 -22677.754} C_VEL
LIN {X 0,Y 179.361,Z 370.957,A -85,B 0,C 180,E1 -22680.002,E2 -22680.002} C_VEL
LIN {X 0,Y 178.868,Z 371.012,A -85,B 0,C 180,E1 -22684.509,E2 -22684.509} C_VEL
LIN {X 0,Y 178.969,Z 371.003,A -85,B 0,C 180,E1 -22689.039,E2 -22689.039} C_VEL
LIN {X 0,Y 178.659,Z 371.04,A -85,B 0,C 180,E1 -22693.654,E2 -22693.654} C_VEL
LIN {X 0,Y 178.632,Z 371.046,A -85,B 0,C 180,E1 -22699.233,E2 -22699.233} C_VEL
LIN {X 0,Y 178.528,Z 371.06,A -85,B 0,C 180,E1 -22705.128,E2 -22705.128} C_VEL
LIN {X 0,Y 178.474,Z 371.063,A -85,B 0,C 180,E1 -22710.794,E2 -22710.794} C_VEL
LIN {X 0,Y 178.48,Z 371.064,A -85,B 0,C 180,E1 -22714.223,E2 -22714.223} C_VEL
LIN {X 0,Y 178.391,Z 371.075,A -85,B 0,C 180,E1 -22719.078,E2 -22719.078} C_VEL
LIN {X 0,Y 178.528,Z 371.055,A -85,B 0,C 180,E1 -22725.123,E2 -22725.123} C_VEL
LIN {X 0,Y 178.652,Z 371.188,A -85,B 0,C 180,E1 -22726.293,E2 -22726.293} C_VEL
LIN {X 0,Y 179.458,Z 375.386,A -85,B 0,C 180,E1 -22731.561,E2 -22731.561} C_VEL
LIN {X 0,Y 179.868,Z 377.509,A -85,B 0,C 180,E1 -22734.123,E2 -22734.123} C_VEL
LIN {X 0,Y 179.634,Z 379.82,A -85,B 0,C 180,E1 -22736.792,E2 -22736.792} C_VEL
LIN {X 0,Y 178.282,Z 384.301,A -85,B 0,C 180,E1 -22741.771,E2 -22741.771} C_VEL
LIN {X 0,Y 177.856,Z 386.007,A -85,B 0,C 180,E1 -22743.662,E2 -22743.662} C_VEL
LIN {X 0,Y 179.209,Z 398.219,A -85,B 0,C 180,E1 -22744.965,E2 -22744.965} C_VEL
LIN {X 0,Y 179.96,Z 409.007,A -85,B 0,C 180,E1 -22746.534,E2 -22746.534} C_VEL
LIN {X 0,Y 180.37,Z 417.397,A -85,B 0,C 180,E1 -22748.058,E2 -22748.058} C_VEL
LIN {X 0,Y 180.522,Z 425.33,A -85,B 0,C 180,E1 -22749.79,E2 -22749.79} C_VEL
LIN {X 0,Y 180.481,Z 432.15,A -85,B 0,C 180,E1 -22751.558,E2 -22751.558} C_VEL
LIN {X 0,Y 179.288,Z 438.577,A -85,B 0,C 180,E1 -22753.492,E2 -22753.492} C_VEL
LIN {X 0,Y 178.217,Z 444.72,A -85,B 0,C 180,E1 -22755.734,E2 -22755.734} C_VEL
LIN {X 0,Y 177.369,Z 449.817,A -85,B 0,C 180,E1 -22757.997,E2 -22757.997} C_VEL
LIN {X 0,Y 176.947,Z 453.11,A -85,B 0,C 180,E1 -22759.707,E2 -22759.707} C_VEL
LIN {X 0,Y 176.509,Z 456.811,A -85,B 0,C 180,E1 -22761.992,E2 -22761.992} C_VEL
LIN {X 0,Y 176.294,Z 460.878,A -85,B 0,C 180,E1 -22765.314,E2 -22765.314} C_VEL
LIN {X 0,Y 176.31,Z 463.086,A -85,B 0,C 180,E1 -22767.718,E2 -22767.718} C_VEL
LIN {X 0,Y 176.415,Z 464.621,A -85,B 0,C 180,E1 -22770.003,E2 -22770.003} C_VEL
LIN {X 0,Y 176.111,Z 465.86,A -85,B 0,C 180,E1 -22773.894,E2 -22773.894} C_VEL
LIN {X 0,Y 176.246,Z 465.896,A -85,B 0,C 180,E1 -22776.874,E2 -22776.874} C_VEL
LIN {X 0,Y 176.869,Z 464.947,A -85,B 0,C 180,E1 -22780.192,E2 -22780.192} C_VEL
LIN {X 0,Y 178.135,Z 462.824,A -85,B 0,C 180,E1 -22783.696,E2 -22783.696} C_VEL
LIN {X 0,Y 180.024,Z 459.614,A -85,B 0,C 180,E1 -22787.028,E2 -22787.028} C_VEL
LIN {X 0,Y 181.876,Z 456.358,A -85,B 0,C 180,E1 -22789.458,E2 -22789.458} C_VEL
LIN {X 0,Y 182.749,Z 453.859,A -85,B 0,C 180,E1 -22791.12,E2 -22791.12} C_VEL
LIN {X 0,Y 182.682,Z 449.317,A -85,B 0,C 180,E1 -22793.886,E2 -22793.886} C_VEL
LIN {X 0,Y 182.449,Z 445.292,A -85,B 0,C 180,E1 -22796.051,E2 -22796.051} C_VEL
LIN {X 0,Y 183.18,Z 440.645,A -85,B 0,C 180,E1 -22798.078,E2 -22798.078} C_VEL
LIN {X 0,Y 185.019,Z 432.926,A -85,B 0,C 180,E1 -22800.853,E2 -22800.853} C_VEL
LIN {X 0,Y 185.898,Z 423.894,A -85,B 0,C 180,E1 -22803.721,E2 -22803.721} C_VEL
LIN {X 0,Y 185.901,Z 415.464,A -85,B 0,C 180,E1 -22806.215,E2 -22806.215} C_VEL
LIN {X 0,Y 185.306,Z 408.895,A -85,B 0,C 180,E1 -22808.163,E2 -22808.163} C_VEL
LIN {X 0,Y 183.827,Z 402.947,A -85,B 0,C 180,E1 -22810.123,E2 -22810.123} C_VEL
LIN {X 0,Y 180.332,Z 395.123,A -85,B 0,C 180,E1 -22813.303,E2 -22813.303} C_VEL
LIN {X 0,Y 179.572,Z 393.373,A -85,B 0,C 180,E1 -22814.046,E2 -22814.046} C_VEL
LIN {X 0,Y 177.391,Z 389.588,A -85,B 0,C 180,E1 -22815.858,E2 -22815.858} C_VEL
LIN {X 0,Y 176.715,Z 387.775,A -85,B 0,C 180,E1 -22816.584,E2 -22816.584} C_VEL
LIN {X 0,Y 173.998,Z 384.037,A -85,B 0,C 180,E1 -22818.975,E2 -22818.975} C_VEL
LIN {X 0,Y 172.989,Z 381.304,A -85,B 0,C 180,E1 -22820.14,E2 -22820.14} C_VEL
LIN {X 0,Y 172.739,Z 379.117,A -85,B 0,C 180,E1 -22825.275,E2 -22825.275} C_VEL
LIN {X 0,Y 172.419,Z 377.293,A -85,B 0,C 180,E1 -22830.714,E2 -22830.714} C_VEL
LIN {X 0,Y 172.23,Z 375.994,A -85,B 0,C 180,E1 -22835.915,E2 -22835.915} C_VEL
LIN {X 0,Y 172.172,Z 375.145,A -85,B 0,C 180,E1 -22840.938,E2 -22840.938} C_VEL
LIN {X 0,Y 172.138,Z 374.723,A -85,B 0,C 180,E1 -22845.818,E2 -22845.818} C_VEL
LIN {X 0,Y 172.335,Z 374.629,A -85,B 0,C 180,E1 -22850.61,E2 -22850.61} C_VEL
LIN {X 0,Y 172.394,Z 374.923,A -85,B 0,C 180,E1 -22855.321,E2 -22855.321} C_VEL
LIN {X 0,Y 172.97,Z 375.408,A -85,B 0,C 180,E1 -22859.998,E2 -22859.998} C_VEL
LIN {X 0,Y 173.794,Z 377.827,A -85,B 0,C 180,E1 -22861.084,E2 -22861.084} C_VEL
LIN {X 0,Y 176.361,Z 381.025,A -85,B 0,C 180,E1 -22863.423,E2 -22863.423} C_VEL
LIN {X 0,Y 177.434,Z 383.426,A -85,B 0,C 180,E1 -22864.541,E2 -22864.541} C_VEL
LIN {X 0,Y 179.406,Z 385.892,A -85,B 0,C 180,E1 -22866.182,E2 -22866.182} C_VEL
LIN {X 0,Y 181.083,Z 389.303,A -85,B 0,C 180,E1 -22867.805,E2 -22867.805} C_VEL
LIN {X 0,Y 184.292,Z 396.337,A -85,B 0,C 180,E1 -22870.99,E2 -22870.99} C_VEL
LIN {X 0,Y 186.447,Z 402.96,A -85,B 0,C 180,E1 -22873.624,E2 -22873.624} C_VEL
LIN {X 0,Y 187.781,Z 410.099,A -85,B 0,C 180,E1 -22876.3,E2 -22876.3} C_VEL
LIN {X 0,Y 188.233,Z 416.854,A -85,B 0,C 180,E1 -22878.783,E2 -22878.783} C_VEL
LIN {X 0,Y 187.836,Z 423.665,A -85,B 0,C 180,E1 -22881.409,E2 -22881.409} C_VEL
LIN {X 0,Y 185.423,Z 428.932,A -85,B 0,C 180,E1 -22883.221,E2 -22883.221} C_VEL
LIN {X 0,Y 183.166,Z 433.258,A -85,B 0,C 180,E1 -22884.962,E2 -22884.962} C_VEL
LIN {X 0,Y 180.23,Z 438.303,A -85,B 0,C 180,E1 -22887.473,E2 -22887.473} C_VEL
LIN {X 0,Y 177.966,Z 441.846,A -85,B 0,C 180,E1 -22889.676,E2 -22889.676} C_VEL
LIN {X 0,Y 175.357,Z 445.472,A -85,B 0,C 180,E1 -22892.681,E2 -22892.681} C_VEL
LIN {X 0,Y 173.211,Z 448.057,A -85,B 0,C 180,E1 -22895.753,E2 -22895.753} C_VEL
LIN {X 0,Y 171.502,Z 449.686,A -85,B 0,C 180,E1 -22898.863,E2 -22898.863} C_VEL
LIN {X 0,Y 170.242,Z 450.416,A -85,B 0,C 180,E1 -22902.001,E2 -22902.001} C_VEL
LIN {X 0,Y 169.39,Z 450.281,A -85,B 0,C 180,E1 -22905.14,E2 -22905.14} C_VEL
LIN {X 0,Y 168.855,Z 449.193,A -85,B 0,C 180,E1 -22908.516,E2 -22908.516} C_VEL
LIN {X 0,Y 168.863,Z 446.847,A -85,B 0,C 180,E1 -22912.253,E2 -22912.253} C_VEL
LIN {X 0,Y 169.357,Z 442.972,A -85,B 0,C 180,E1 -22916.09,E2 -22916.09} C_VEL
LIN {X 0,Y 169.977,Z 439.247,A -85,B 0,C 180,E1 -22918.819,E2 -22918.819} C_VEL
LIN {X 0,Y 170.909,Z 434.097,A -85,B 0,C 180,E1 -22921.775,E2 -22921.775} C_VEL
LIN {X 0,Y 172.179,Z 427.689,A -85,B 0,C 180,E1 -22924.682,E2 -22924.682} C_VEL
LIN {X 0,Y 173.437,Z 420.786,A -85,B 0,C 180,E1 -22927.202,E2 -22927.202} C_VEL
LIN {X 0,Y 175.106,Z 412.088,A -85,B 0,C 180,E1 -22929.744,E2 -22929.744} C_VEL
LIN {X 0,Y 176.084,Z 405.163,A -85,B 0,C 180,E1 -22931.376,E2 -22931.376} C_VEL
LIN {X 0,Y 174.948,Z 395.826,A -85,B 0,C 180,E1 -22933.365,E2 -22933.365} C_VEL
LIN {X 0,Y 173.471,Z 386.217,A -85,B 0,C 180,E1 -22935.029,E2 -22935.029} C_VEL
LIN {X 0,Y 171.67,Z 376.641,A -85,B 0,C 180,E1 -22936.382,E2 -22936.382} C_VEL
LIN {X 0,Y 170.648,Z 372.043,A -85,B 0,C 180,E1 -22936.981,E2 -22936.981} C_VEL
LIN {X 0,Y 171.28,Z 371.964,A -85,B 0,C 180,E1 -22940.55,E2 -22940.55} C_VEL
LIN {X 0,Y 171.615,Z 371.922,A -85,B 0,C 180,E1 -22942.94,E2 -22942.94} C_VEL
LIN {X 0,Y 172.074,Z 371.865,A -85,B 0,C 180,E1 -22947.656,E2 -22947.656} C_VEL
LIN {X 0,Y 172.323,Z 371.835,A -85,B 0,C 180,E1 -22949.997,E2 -22949.997} C_VEL
LIN {X 0,Y 171.819,Z 371.894,A -85,B 0,C 180,E1 -22954.689,E2 -22954.689} C_VEL
LIN {X 0,Y 171.901,Z 371.884,A -85,B 0,C 180,E1 -22959.409,E2 -22959.409} C_VEL
LIN {X 0,Y 171.6,Z 371.922,A -85,B 0,C 180,E1 -22964.222,E2 -22964.222} C_VEL
LIN {X 0,Y 171.534,Z 371.927,A -85,B 0,C 180,E1 -22969.56,E2 -22969.56} C_VEL
LIN {X 0,Y 171.458,Z 371.939,A -85,B 0,C 180,E1 -22975.615,E2 -22975.615} C_VEL
LIN {X 0,Y 171.43,Z 371.941,A -85,B 0,C 180,E1 -22980.585,E2 -22980.585} C_VEL
LIN {X 0,Y 171.397,Z 371.946,A -85,B 0,C 180,E1 -22985.03,E2 -22985.03} C_VEL
LIN {X 0,Y 171.434,Z 371.941,A -85,B 0,C 180,E1 -22988.844,E2 -22988.844} C_VEL
LIN {X 0,Y 171.443,Z 371.937,A -85,B 0,C 180,E1 -22994.173,E2 -22994.173} C_VEL
LIN {X 0,Y 171.423,Z 371.945,A -85,B 0,C 180,E1 -22999.01,E2 -22999.01} C_VEL
LIN {X 0,Y 171.43,Z 371.94,A -85,B 0,C 180,E1 -23002.056,E2 -23002.056} C_VEL
LIN {X 0,Y 171.407,Z 371.945,A -85,B 0,C 180,E1 -23007.793,E2 -23007.793} C_VEL
LIN {X 0,Y 171.437,Z 371.939,A -85,B 0,C 180,E1 -23010.535,E2 -23010.535} C_VEL
LIN {X 0,Y 171.464,Z 371.938,A -85,B 0,C 180,E1 -23015.805,E2 -23015.805} C_VEL
LIN {X 0,Y 171.6,Z 371.92,A -85,B 0,C 180,E1 -23020.877,E2 -23020.877} C_VEL
LIN {X 0,Y 171.605,Z 371.92,A -85,B 0,C 180,E1 -23025.778,E2 -23025.778} C_VEL
LIN {X 0,Y 171.9,Z 371.885,A -85,B 0,C 180,E1 -23030.59,E2 -23030.59} C_VEL
LIN {X 0,Y 171.816,Z 371.891,A -85,B 0,C 180,E1 -23035.31,E2 -23035.31} C_VEL
LIN {X 0,Y 172.323,Z 371.834,A -85,B 0,C 180,E1 -23040.002,E2 -23040.002} C_VEL
LIN {X 0,Y 171.817,Z 371.89,A -85,B 0,C 180,E1 -23044.695,E2 -23044.695} C_VEL
LIN {X 0,Y 171.896,Z 371.886,A -85,B 0,C 180,E1 -23049.415,E2 -23049.415} C_VEL
LIN {X 0,Y 171.578,Z 371.923,A -85,B 0,C 180,E1 -23054.229,E2 -23054.229} C_VEL
LIN {X 0,Y 171.551,Z 371.926,A -85,B 0,C 180,E1 -23059.577,E2 -23059.577} C_VEL
LIN {X 0,Y 171.463,Z 371.939,A -85,B 0,C 180,E1 -23065.62,E2 -23065.62} C_VEL
LIN {X 0,Y 171.437,Z 371.939,A -85,B 0,C 180,E1 -23070.59,E2 -23070.59} C_VEL
LIN {X 0,Y 171.388,Z 371.949,A -85,B 0,C 180,E1 -23075.038,E2 -23075.038} C_VEL
LIN {X 0,Y 171.353,Z 371.95,A -85,B 0,C 180,E1 -23078.811,E2 -23078.811} C_VEL
LIN {X 0,Y 171.401,Z 371.944,A -85,B 0,C 180,E1 -23084.194,E2 -23084.194} C_VEL
LIN {X 0,Y 171.607,Z 372.028,A -85,B 0,C 180,E1 -23086.212,E2 -23086.212} C_VEL
LIN {X 0,Y 172.524,Z 376.747,A -85,B 0,C 180,E1 -23092.339,E2 -23092.339} C_VEL
LIN {X 0,Y 172.727,Z 379.122,A -85,B 0,C 180,E1 -23095.279,E2 -23095.279} C_VEL
LIN {X 0,Y 172.167,Z 381.399,A -85,B 0,C 180,E1 -23097.953,E2 -23097.953} C_VEL
LIN {X 0,Y 170.868,Z 385.714,A -85,B 0,C 180,E1 -23102.938,E2 -23102.938} C_VEL
LIN {X 0,Y 172.246,Z 398.123,A -85,B 0,C 180,E1 -23104.338,E2 -23104.338} C_VEL
LIN {X 0,Y 172.956,Z 408.03,A -85,B 0,C 180,E1 -23105.832,E2 -23105.832} C_VEL
LIN {X 0,Y 173.328,Z 416.213,A -85,B 0,C 180,E1 -23107.347,E2 -23107.347} C_VEL
LIN {X 0,Y 173.474,Z 424.669,A -85,B 0,C 180,E1 -23109.241,E2 -23109.241} C_VEL
LIN {X 0,Y 173.46,Z 431.573,A -85,B 0,C 180,E1 -23111.09,E2 -23111.09} C_VEL
LIN {X 0,Y 172.472,Z 437.202,A -85,B 0,C 180,E1 -23112.82,E2 -23112.82} C_VEL
LIN {X 0,Y 171.327,Z 443.508,A -85,B 0,C 180,E1 -23115.148,E2 -23115.148} C_VEL
LIN {X 0,Y 170.403,Z 448.747,A -85,B 0,C 180,E1 -23117.498,E2 -23117.498} C_VEL
LIN {X 0,Y 169.693,Z 454.074,A -85,B 0,C 180,E1 -23120.467,E2 -23120.467} C_VEL
LIN {X 0,Y 169.343,Z 457.499,A -85,B 0,C 180,E1 -23122.851,E2 -23122.851} C_VEL
LIN {X 0,Y 169.218,Z 460.457,A -85,B 0,C 180,E1 -23125.418,E2 -23125.418} C_VEL
LIN {X 0,Y 169.231,Z 462.484,A -85,B 0,C 180,E1 -23127.623,E2 -23127.623} C_VEL
LIN {X 0,Y 169.351,Z 464.047,A -85,B 0,C 180,E1 -23130.003,E2 -23130.003} C_VEL
LIN {X 0,Y 169.03,Z 465.43,A -85,B 0,C 180,E1 -23133.704,E2 -23133.704} C_VEL
LIN {X 0,Y 169.178,Z 465.607,A -85,B 0,C 180,E1 -23137.162,E2 -23137.162} C_VEL
LIN {X 0,Y 169.611,Z 465.177,A -85,B 0,C 180,E1 -23139.543,E2 -23139.543} C_VEL
LIN {X 0,Y 170.292,Z 464.189,A -85,B 0,C 180,E1 -23141.912,E2 -23141.912} C_VEL
LIN {X 0,Y 171.233,Z 462.755,A -85,B 0,C 180,E1 -23144.259,E2 -23144.259} C_VEL
LIN {X 0,Y 173.233,Z 459.676,A -85,B 0,C 180,E1 -23147.717,E2 -23147.717} C_VEL
LIN {X 0,Y 175.98,Z 455.383,A -85,B 0,C 180,E1 -23151.068,E2 -23151.068} C_VEL
LIN {X 0,Y 179.383,Z 449.59,A -85,B 0,C 180,E1 -23154.294,E2 -23154.294} C_VEL
LIN {X 0,Y 181.723,Z 444.852,A -85,B 0,C 180,E1 -23156.411,E2 -23156.411} C_VEL
LIN {X 0,Y 183.18,Z 440.645,A -85,B 0,C 180,E1 -23158.078,E2 -23158.078} C_VEL
LIN {X 0,Y 183.613,Z 437.125,A -85,B 0,C 180,E1 -23159.549,E2 -23159.549} C_VEL
LIN {X 0,Y 183.013,Z 433.799,A -85,B 0,C 180,E1 -23161.079,E2 -23161.079} C_VEL
LIN {X 0,Y 180.821,Z 427.093,A -85,B 0,C 180,E1 -23164.16,E2 -23164.16} C_VEL
LIN {X 0,Y 180.245,Z 421.902,A -85,B 0,C 180,E1 -23166.094,E2 -23166.094} C_VEL
LIN {X 0,Y 180.217,Z 415.138,A -85,B 0,C 180,E1 -23168.254,E2 -23168.254} C_VEL
LIN {X 0,Y 179.582,Z 409.968,A -85,B 0,C 180,E1 -23170.017,E2 -23170.017} C_VEL
LIN {X 0,Y 177.901,Z 404.479,A -85,B 0,C 180,E1 -23172.193,E2 -23172.193} C_VEL
LIN {X 0,Y 175.732,Z 399.201,A -85,B 0,C 180,E1 -23174.579,E2 -23174.579} C_VEL
LIN {X 0,Y 172.732,Z 392.989,A -85,B 0,C 180,E1 -23177.825,E2 -23177.825} C_VEL
LIN {X 0,Y 170.381,Z 388.887,A -85,B 0,C 180,E1 -23180.311,E2 -23180.311} C_VEL
LIN {X 0,Y 169.744,Z 387.238,A -85,B 0,C 180,E1 -23181.187,E2 -23181.187} C_VEL
LIN {X 0,Y 167.016,Z 383.602,A -85,B 0,C 180,E1 -23184.421,E2 -23184.421} C_VEL
LIN {X 0,Y 165.678,Z 380.237,A -85,B 0,C 180,E1 -23186.768,E2 -23186.768} C_VEL
LIN {X 0,Y 165.582,Z 379.398,A -85,B 0,C 180,E1 -23189.378,E2 -23189.378} C_VEL
LIN {X 0,Y 165.359,Z 377.983,A -85,B 0,C 180,E1 -23194.846,E2 -23194.846} C_VEL
LIN {X 0,Y 165.316,Z 377.029,A -85,B 0,C 180,E1 -23200.115,E2 -23200.115} C_VEL
LIN {X 0,Y 165.249,Z 376.524,A -85,B 0,C 180,E1 -23205.214,E2 -23205.214} C_VEL
LIN {X 0,Y 165.416,Z 376.38,A -85,B 0,C 180,E1 -23210.213,E2 -23210.213} C_VEL
LIN {X 0,Y 165.507,Z 376.585,A -85,B 0,C 180,E1 -23213.292,E2 -23213.292} C_VEL
LIN {X 0,Y 166.525,Z 378.905,A -85,B 0,C 180,E1 -23215.156,E2 -23215.156} C_VEL
LIN {X 0,Y 170.092,Z 382.037,A -85,B 0,C 180,E1 -23219.331,E2 -23219.331} C_VEL
LIN {X 0,Y 171.512,Z 385.052,A -85,B 0,C 180,E1 -23221.172,E2 -23221.172} C_VEL
LIN {X 0,Y 172.629,Z 386.467,A -85,B 0,C 180,E1 -23222.331,E2 -23222.331} C_VEL
LIN {X 0,Y 174.586,Z 390.312,A -85,B 0,C 180,E1 -23224.616,E2 -23224.616} C_VEL
LIN {X 0,Y 175.745,Z 392.053,A -85,B 0,C 180,E1 -23225.735,E2 -23225.735} C_VEL
LIN {X 0,Y 178.582,Z 398.525,A -85,B 0,C 180,E1 -23229.055,E2 -23229.055} C_VEL
LIN {X 0,Y 180.537,Z 404.445,A -85,B 0,C 180,E1 -23231.79,E2 -23231.79} C_VEL
LIN {X 0,Y 181.655,Z 409.897,A -85,B 0,C 180,E1 -23234.048,E2 -23234.048} C_VEL
LIN {X 0,Y 182.259,Z 416.685,A -85,B 0,C 180,E1 -23236.808,E2 -23236.808} C_VEL
LIN {X 0,Y 182.018,Z 422.473,A -85,B 0,C 180,E1 -23239.157,E2 -23239.157} C_VEL
LIN {X 0,Y 181.685,Z 425.336,A -85,B 0,C 180,E1 -23240.371,E2 -23240.371} C_VEL
LIN {X 0,Y 179.968,Z 428.983,A -85,B 0,C 180,E1 -23241.705,E2 -23241.705} C_VEL
LIN {X 0,Y 176.906,Z 434.405,A -85,B 0,C 180,E1 -23243.969,E2 -23243.969} C_VEL
LIN {X 0,Y 173.999,Z 439.004,A -85,B 0,C 180,E1 -23246.376,E2 -23246.376} C_VEL
LIN {X 0,Y 171.9,Z 442.087,A -85,B 0,C 180,E1 -23248.356,E2 -23248.356} C_VEL
LIN {X 0,Y 169.002,Z 445.791,A -85,B 0,C 180,E1 -23251.513,E2 -23251.513} C_VEL
LIN {X 0,Y 166.674,Z 448.383,A -85,B 0,C 180,E1 -23254.686,E2 -23254.686} C_VEL
LIN {X 0,Y 165.614,Z 449.469,A -85,B 0,C 180,E1 -23256.445,E2 -23256.445} C_VEL
LIN {X 0,Y 163.821,Z 450.665,A -85,B 0,C 180,E1 -23260.05,E2 -23260.05} C_VEL
LIN {X 0,Y 162.608,Z 450.758,A -85,B 0,C 180,E1 -23263.747,E2 -23263.747} C_VEL
LIN {X 0,Y 162.098,Z 450.34,A -85,B 0,C 180,E1 -23266.072,E2 -23266.072} C_VEL
LIN {X 0,Y 161.718,Z 448.958,A -85,B 0,C 180,E1 -23269.313,E2 -23269.313} C_VEL
LIN {X 0,Y 161.785,Z 446.723,A -85,B 0,C 180,E1 -23272.54,E2 -23272.54} C_VEL
LIN {X 0,Y 162.173,Z 443.62,A -85,B 0,C 180,E1 -23275.707,E2 -23275.707} C_VEL
LIN {X 0,Y 162.845,Z 439.596,A -85,B 0,C 180,E1 -23278.806,E2 -23278.806} C_VEL
LIN {X 0,Y 163.785,Z 434.555,A -85,B 0,C 180,E1 -23281.832,E2 -23281.832} C_VEL
LIN {X 0,Y 165.034,Z 428.341,A -85,B 0,C 180,E1 -23284.792,E2 -23284.792} C_VEL
LIN {X 0,Y 166.272,Z 421.806,A -85,B 0,C 180,E1 -23287.31,E2 -23287.31} C_VEL
LIN {X 0,Y 167.851,Z 413.839,A -85,B 0,C 180,E1 -23289.789,E2 -23289.789} C_VEL
LIN {X 0,Y 169.085,Z 405.747,A -85,B 0,C 180,E1 -23291.833,E2 -23291.833} C_VEL
LIN {X 0,Y 167.81,Z 394.959,A -85,B 0,C 180,E1 -23294.2,E2 -23294.2} C_VEL
LIN {X 0,Y 166.261,Z 385.246,A -85,B 0,C 180,E1 -23295.93,E2 -23295.93} C_VEL
LIN {X 0,Y 164.46,Z 375.964,A -85,B 0,C 180,E1 -23297.268,E2 -23297.268} C_VEL
LIN {X 0,Y 163.722,Z 372.904,A -85,B 0,C 180,E1 -23297.689,E2 -23297.689} C_VEL
LIN {X 0,Y 164.501,Z 372.81,A -85,B 0,C 180,E1 -23302.633,E2 -23302.633} C_VEL
LIN {X 0,Y 165.018,Z 372.744,A -85,B 0,C 180,E1 -23307.556,E2 -23307.556} C_VEL
